LIN {X 79.043,Y 42.209,Z 71.697,A 180.000,B 0.000,C 180.000} C_DIS
LIN {X 79.064,Y 42.285,Z 71.694,A 180.000,B 0.000,C 180.000} C_DIS
LIN {X 79.085,Y 42.362,Z 71.691,A 180.000,B 0.000,C 180.000} C_DIS
LIN {X 79.105,Y 42.438,Z 71.689,A 180.000,B 0.000,C 180.000} C_DIS
LIN {X 79.126,Y 42.514,Z 71.686,A 180.000,B 0.000,C 180.000} C_DIS
LIN {X 79.147,Y 42.590,Z 71.683,A 180.000,B 0.000,C 180.000} C_DIS
LIN {X 79.167,Y 42.666,Z 71.680,A 180.000,B 0.000,C 180.000} C_DIS
LIN {X 79.188,Y 42.742,Z 71.678,A 180.000,B 0.000,C 180.000} C_DIS
LIN {X 79.209,Y 42.818,Z 71.675,A 180.000,B 0.000,C 180.000} C_DIS
LIN {X 79.230,Y 42.894,Z 71.672,A 180.000,B 0.000,C 180.000} C_DIS
LIN {X 79.250,Y 42.971,Z 71.670,A 180.000,B 0.000,C 180.000} C_DIS
LIN {X 79.271,Y 43.047,Z 71.667,A 180.000,B 0.000,C 180.000} C_DIS
LIN {X 79.292,Y 43.123,Z 71.665,A 180.000,B 0.000,C 180.000} C_DIS
LIN {X 79.313,Y 43.199,Z 71.662,A 180.000,B 0.000,C 180.000} C_DIS
LIN {X 79.334,Y 43.275,Z 71.659,A 180.000,B 0.000,C 180.000} C_DIS
LIN {X 79.355,Y 43.351,Z 71.657,A 180.000,B 0.000,C 180.000} C_DIS
LIN {X 79.376,Y 43.427,Z 71.654,A 180.000,B 0.000,C 180.000} C_DIS
LIN {X 79.397,Y 43.503,Z 71.652,A 180.000,B 0.000,C 180.000} C_DIS
LIN {X 79.418,Y 43.579,Z 71.649,A 180.000,B 0.000,C 180.000} C_DIS
LIN {X 79.439,Y 43.655,Z 71.647,A 180.000,B 0.000,C 180.000} C_DIS
LIN {X 79.481,Y 43.807,Z 71.642,A 180.000,B 0.000,C 180.000} C_DIS
LIN {X 79.523,Y 43.959,Z 71.637,A 180.000,B 0.000,C 180.000} C_DIS
LIN {X 79.565,Y 44.111,Z 71.632,A 180.000,B 0.000,C 180.000} C_DIS
LIN {X 79.608,Y 44.263,Z 71.627,A 180.000,B 0.000,C 180.000} C_DIS
LIN {X 79.650,Y 44.415,Z 71.623,A 180.000,B 0.000,C 180.000} C_DIS
LIN {X 79.693,Y 44.566,Z 71.618,A 180.000,B 0.000,C 180.000} C_DIS
LIN {X 79.736,Y 44.718,Z 71.613,A 180.000,B 0.000,C 180.000} C_DIS
LIN {X 79.779,Y 44.870,Z 71.609,A 180.000,B 0.000,C 180.000} C_DIS
LIN {X 79.822,Y 45.022,Z 71.604,A 180.000,B 0.000,C 180.000} C_DIS
LIN {X 79.865,Y 45.173,Z 71.600,A 180.000,B 0.000,C 180.000} C_DIS
LIN {X 79.908,Y 45.325,Z 71.596,A 180.000,B 0.000,C 180.000} C_DIS
LIN {X 79.952,Y 45.477,Z 71.592,A 180.000,B 0.000,C 180.000} C_DIS
LIN {X 79.995,Y 45.628,Z 71.588,A 180.000,B 0.000,C 180.000} C_DIS
LIN {X 80.039,Y 45.780,Z 71.584,A 180.000,B 0.000,C 180.000} C_DIS
LIN {X 80.083,Y 45.931,Z 71.580,A 180.000,B 0.000,C 180.000} C_DIS
LIN {X 80.127,Y 46.082,Z 71.576,A 180.000,B 0.000,C 180.000} C_DIS
LIN {X 80.171,Y 46.234,Z 71.572,A 180.000,B 0.000,C 180.000} C_DIS
LIN {X 80.215,Y 46.385,Z 71.568,A 180.000,B 0.000,C 180.000} C_DIS
LIN {X 80.259,Y 46.536,Z 71.565,A 180.000,B 0.000,C 180.000} C_DIS
LIN {X 80.304,Y 46.688,Z 71.561,A 180.000,B 0.000,C 180.000} C_DIS
LIN {X 80.348,Y 46.839,Z 71.558,A 180.000,B 0.000,C 180.000} C_DIS
LIN {X 80.393,Y 46.990,Z 71.554,A 180.000,B 0.000,C 180.000} C_DIS
LIN {X 80.438,Y 47.141,Z 71.551,A 180.000,B 0.000,C 180.000} C_DIS
LIN {X 80.483,Y 47.292,Z 71.548,A 180.000,B 0.000,C 180.000} C_DIS
LIN {X 80.528,Y 47.443,Z 71.545,A 180.000,B 0.000,C 180.000} C_DIS
LIN {X 80.574,Y 47.594,Z 71.542,A 180.000,B 0.000,C 180.000} C_DIS
LIN {X 80.619,Y 47.745,Z 71.539,A 180.000,B 0.000,C 180.000} C_DIS
LIN {X 80.665,Y 47.895,Z 71.536,A 180.000,B 0.000,C 180.000} C_DIS
LIN {X 80.711,Y 48.046,Z 71.533,A 180.000,B 0.000,C 180.000} C_DIS
LIN {X 80.757,Y 48.197,Z 71.531,A 180.000,B 0.000,C 180.000} C_DIS
LIN {X 80.803,Y 48.348,Z 71.528,A 180.000,B 0.000,C 180.000} C_DIS
LIN {X 80.896,Y 48.649,Z 71.524,A 180.000,B 0.000,C 180.000} C_DIS
LIN {X 80.989,Y 48.950,Z 71.519,A 180.000,B 0.000,C 180.000} C_DIS
LIN {X 81.084,Y 49.250,Z 71.515,A 180.000,B 0.000,C 180.000} C_DIS
LIN {X 81.178,Y 49.551,Z 71.512,A 180.000,B 0.000,C 180.000} C_DIS
LIN {X 81.274,Y 49.851,Z 71.509,A 180.000,B 0.000,C 180.000} C_DIS
LIN {X 81.370,Y 50.151,Z 71.506,A 180.000,B 0.000,C 180.000} C_DIS
LIN {X 81.467,Y 50.451,Z 71.504,A 180.000,B 0.000,C 180.000} C_DIS
LIN {X 81.564,Y 50.750,Z 71.502,A 180.000,B 0.000,C 180.000} C_DIS
LIN {X 81.663,Y 51.049,Z 71.501,A 180.000,B 0.000,C 180.000} C_DIS
LIN {X 81.762,Y 51.348,Z 71.500,A 180.000,B 0.000,C 180.000} C_DIS
LIN {X 81.862,Y 51.647,Z 71.500,A 180.000,B 0.000,C 180.000} C_DIS
LIN {X 81.868,Y 51.663,Z 71.500,A 180.000,B 0.000,C 180.000} C_DIS
; Cutting Move Starts
LIN {X 84.885,Y 60.606,Z 71.500,A 180.000,B 0.000,C 180.000} C_DIS
LIN {X 84.919,Y 60.703,Z 71.500,A 180.000,B 0.000,C 180.000} C_DIS
LIN {X 84.952,Y 60.785,Z 71.500,A 180.000,B 0.000,C 180.000} C_DIS
LIN {X 85.035,Y 60.964,Z 71.500,A 180.000,B 0.000,C 180.000} C_DIS
LIN {X 85.098,Y 61.079,Z 71.500,A 180.000,B 0.000,C 180.000} C_DIS
LIN {X 85.136,Y 61.143,Z 71.500,A 180.000,B 0.000,C 180.000} C_DIS
LIN {X 85.258,Y 61.321,Z 71.500,A 180.000,B 0.000,C 180.000} C_DIS
LIN {X 85.276,Y 61.345,Z 71.500,A 180.000,B 0.000,C 180.000} C_DIS
LIN {X 85.406,Y 61.500,Z 71.500,A 180.000,B 0.000,C 180.000} C_DIS
LIN {X 85.455,Y 61.553,Z 71.500,A 180.000,B 0.000,C 180.000} C_DIS
LIN {X 85.585,Y 61.679,Z 71.500,A 180.000,B 0.000,C 180.000} C_DIS
LIN {X 85.634,Y 61.722,Z 71.500,A 180.000,B 0.000,C 180.000} C_DIS
LIN {X 85.808,Y 61.858,Z 71.500,A 180.000,B 0.000,C 180.000} C_DIS
LIN {X 85.813,Y 61.861,Z 71.500,A 180.000,B 0.000,C 180.000} C_DIS
LIN {X 85.992,Y 61.977,Z 71.500,A 180.000,B 0.000,C 180.000} C_DIS
LIN {X 86.099,Y 62.036,Z 71.500,A 180.000,B 0.000,C 180.000} C_DIS
LIN {X 86.170,Y 62.073,Z 71.500,A 180.000,B 0.000,C 180.000} C_DIS
LIN {X 86.349,Y 62.151,Z 71.500,A 180.000,B 0.000,C 180.000} C_DIS
LIN {X 86.528,Y 62.213,Z 71.500,A 180.000,B 0.000,C 180.000} C_DIS
LIN {X 86.536,Y 62.215,Z 71.500,A 180.000,B 0.000,C 180.000} C_DIS
LIN {X 86.707,Y 62.260,Z 71.500,A 180.000,B 0.000,C 180.000} C_DIS
LIN {X 86.885,Y 62.294,Z 71.500,A 180.000,B 0.000,C 180.000} C_DIS
LIN {X 86.975,Y 62.306,Z 71.500,A 180.000,B 0.000,C 180.000} C_DIS
LIN {X 87.064,Y 62.314,Z 71.500,A 180.000,B 0.000,C 180.000} C_DIS
LIN {X 87.154,Y 62.320,Z 71.500,A 180.000,B 0.000,C 180.000} C_DIS
LIN {X 87.243,Y 62.322,Z 71.500,A 180.000,B 0.000,C 180.000} C_DIS
LIN {X 87.332,Y 62.321,Z 71.500,A 180.000,B 0.000,C 180.000} C_DIS
LIN {X 87.422,Y 62.317,Z 71.500,A 180.000,B 0.000,C 180.000} C_DIS
LIN {X 87.511,Y 62.309,Z 71.500,A 180.000,B 0.000,C 180.000} C_DIS
LIN {X 87.601,Y 62.298,Z 71.500,A 180.000,B 0.000,C 180.000} C_DIS
LIN {X 87.690,Y 62.284,Z 71.500,A 180.000,B 0.000,C 180.000} C_DIS
LIN {X 87.779,Y 62.267,Z 71.500,A 180.000,B 0.000,C 180.000} C_DIS
LIN {X 87.869,Y 62.246,Z 71.500,A 180.000,B 0.000,C 180.000} C_DIS
LIN {X 87.958,Y 62.222,Z 71.500,A 180.000,B 0.000,C 180.000} C_DIS
LIN {X 87.981,Y 62.215,Z 71.500,A 180.000,B 0.000,C 180.000} C_DIS
LIN {X 88.137,Y 62.164,Z 71.500,A 180.000,B 0.000,C 180.000} C_DIS
LIN {X 96.464,Y 59.355,Z 71.500,A 180.000,B 0.000,C 180.000} C_DIS
LIN {X 96.539,Y 59.329,Z 71.500,A 180.000,B 0.000,C 180.000} C_DIS
LIN {X 96.718,Y 59.257,Z 71.500,A 180.000,B 0.000,C 180.000} C_DIS
LIN {X 96.883,Y 59.176,Z 71.500,A 180.000,B 0.000,C 180.000} C_DIS
LIN {X 96.897,Y 59.169,Z 71.500,A 180.000,B 0.000,C 180.000} C_DIS
LIN {X 97.075,Y 59.061,Z 71.500,A 180.000,B 0.000,C 180.000} C_DIS
LIN {X 97.167,Y 58.997,Z 71.500,A 180.000,B 0.000,C 180.000} C_DIS
LIN {X 97.254,Y 58.931,Z 71.500,A 180.000,B 0.000,C 180.000} C_DIS
LIN {X 97.385,Y 58.819,Z 71.500,A 180.000,B 0.000,C 180.000} C_DIS
LIN {X 97.433,Y 58.774,Z 71.500,A 180.000,B 0.000,C 180.000} C_DIS
LIN {X 97.562,Y 58.640,Z 71.500,A 180.000,B 0.000,C 180.000} C_DIS
LIN {X 97.612,Y 58.582,Z 71.500,A 180.000,B 0.000,C 180.000} C_DIS
LIN {X 97.707,Y 58.461,Z 71.500,A 180.000,B 0.000,C 180.000} C_DIS
LIN {X 97.790,Y 58.341,Z 71.500,A 180.000,B 0.000,C 180.000} C_DIS
LIN {X 97.828,Y 58.282,Z 71.500,A 180.000,B 0.000,C 180.000} C_DIS
LIN {X 97.928,Y 58.103,Z 71.500,A 180.000,B 0.000,C 180.000} C_DIS
LIN {X 97.969,Y 58.017,Z 71.500,A 180.000,B 0.000,C 180.000} C_DIS
LIN {X 98.009,Y 57.925,Z 71.500,A 180.000,B 0.000,C 180.000} C_DIS
LIN {X 98.075,Y 57.746,Z 71.500,A 180.000,B 0.000,C 180.000} C_DIS
LIN {X 98.125,Y 57.567,Z 71.500,A 180.000,B 0.000,C 180.000} C_DIS
LIN {X 98.148,Y 57.466,Z 71.500,A 180.000,B 0.000,C 180.000} C_DIS
LIN {X 98.162,Y 57.388,Z 71.500,A 180.000,B 0.000,C 180.000} C_DIS
LIN {X 98.186,Y 57.210,Z 71.500,A 180.000,B 0.000,C 180.000} C_DIS
LIN {X 98.196,Y 57.031,Z 71.500,A 180.000,B 0.000,C 180.000} C_DIS
LIN {X 98.193,Y 56.852,Z 71.500,A 180.000,B 0.000,C 180.000} C_DIS
LIN {X 98.178,Y 56.673,Z 71.500,A 180.000,B 0.000,C 180.000} C_DIS
LIN {X 98.150,Y 56.495,Z 71.500,A 180.000,B 0.000,C 180.000} C_DIS
LIN {X 98.148,Y 56.485,Z 71.500,A 180.000,B 0.000,C 180.000} C_DIS
LIN {X 98.108,Y 56.316,Z 71.500,A 180.000,B 0.000,C 180.000} C_DIS
LIN {X 98.052,Y 56.137,Z 71.500,A 180.000,B 0.000,C 180.000} C_DIS
LIN {X 91.712,Y 37.344,Z 71.500,A 180.000,B 0.000,C 180.000} C_DIS
LIN {X 91.659,Y 37.187,Z 71.500,A 180.000,B 0.000,C 180.000} C_DIS
LIN {X 91.588,Y 37.009,Z 71.500,A 180.000,B 0.000,C 180.000} C_DIS
LIN {X 91.533,Y 36.894,Z 71.500,A 180.000,B 0.000,C 180.000} C_DIS
LIN {X 91.500,Y 36.830,Z 71.500,A 180.000,B 0.000,C 180.000} C_DIS
LIN {X 91.392,Y 36.651,Z 71.500,A 180.000,B 0.000,C 180.000} C_DIS
LIN {X 91.355,Y 36.595,Z 71.500,A 180.000,B 0.000,C 180.000} C_DIS
LIN {X 91.263,Y 36.472,Z 71.500,A 180.000,B 0.000,C 180.000} C_DIS
LIN {X 91.176,Y 36.368,Z 71.500,A 180.000,B 0.000,C 180.000} C_DIS
LIN {X 91.107,Y 36.294,Z 71.500,A 180.000,B 0.000,C 180.000} C_DIS
LIN {X 90.997,Y 36.186,Z 71.500,A 180.000,B 0.000,C 180.000} C_DIS
LIN {X 90.917,Y 36.115,Z 71.500,A 180.000,B 0.000,C 180.000} C_DIS
LIN {X 90.818,Y 36.036,Z 71.500,A 180.000,B 0.000,C 180.000} C_DIS
LIN {X 90.677,Y 35.936,Z 71.500,A 180.000,B 0.000,C 180.000} C_DIS
LIN {X 90.640,Y 35.912,Z 71.500,A 180.000,B 0.000,C 180.000} C_DIS
LIN {X 90.461,Y 35.809,Z 71.500,A 180.000,B 0.000,C 180.000} C_DIS
LIN {X 90.356,Y 35.757,Z 71.500,A 180.000,B 0.000,C 180.000} C_DIS
LIN {X 90.282,Y 35.724,Z 71.500,A 180.000,B 0.000,C 180.000} C_DIS
LIN {X 90.103,Y 35.656,Z 71.500,A 180.000,B 0.000,C 180.000} C_DIS
LIN {X 89.925,Y 35.603,Z 71.500,A 180.000,B 0.000,C 180.000} C_DIS
LIN {X 89.819,Y 35.578,Z 71.500,A 180.000,B 0.000,C 180.000} C_DIS
LIN {X 89.746,Y 35.564,Z 71.500,A 180.000,B 0.000,C 180.000} C_DIS
LIN {X 89.567,Y 35.539,Z 71.500,A 180.000,B 0.000,C 180.000} C_DIS
LIN {X 89.388,Y 35.526,Z 71.500,A 180.000,B 0.000,C 180.000} C_DIS
LIN {X 89.209,Y 35.526,Z 71.500,A 180.000,B 0.000,C 180.000} C_DIS
LIN {X 89.031,Y 35.540,Z 71.500,A 180.000,B 0.000,C 180.000} C_DIS
LIN {X 88.852,Y 35.566,Z 71.500,A 180.000,B 0.000,C 180.000} C_DIS
LIN {X 88.788,Y 35.578,Z 71.500,A 180.000,B 0.000,C 180.000} C_DIS
LIN {X 88.673,Y 35.605,Z 71.500,A 180.000,B 0.000,C 180.000} C_DIS
LIN {X 88.494,Y 35.659,Z 71.500,A 180.000,B 0.000,C 180.000} C_DIS
LIN {X 80.092,Y 38.494,Z 71.500,A 180.000,B 0.000,C 180.000} C_DIS
LIN {X 80.003,Y 38.525,Z 71.500,A 180.000,B 0.000,C 180.000} C_DIS
LIN {X 79.913,Y 38.560,Z 71.500,A 180.000,B 0.000,C 180.000} C_DIS
LIN {X 79.848,Y 38.587,Z 71.500,A 180.000,B 0.000,C 180.000} C_DIS
LIN {X 79.783,Y 38.618,Z 71.500,A 180.000,B 0.000,C 180.000} C_DIS
LIN {X 79.735,Y 38.642,Z 71.500,A 180.000,B 0.000,C 180.000} C_DIS
LIN {X 79.645,Y 38.689,Z 71.500,A 180.000,B 0.000,C 180.000} C_DIS
LIN {X 79.556,Y 38.742,Z 71.500,A 180.000,B 0.000,C 180.000} C_DIS
LIN {X 79.471,Y 38.796,Z 71.500,A 180.000,B 0.000,C 180.000} C_DIS
LIN {X 79.377,Y 38.863,Z 71.500,A 180.000,B 0.000,C 180.000} C_DIS
LIN {X 79.307,Y 38.917,Z 71.500,A 180.000,B 0.000,C 180.000} C_DIS
LIN {X 79.236,Y 38.975,Z 71.500,A 180.000,B 0.000,C 180.000} C_DIS
LIN {X 79.198,Y 39.008,Z 71.500,A 180.000,B 0.000,C 180.000} C_DIS
LIN {X 79.124,Y 39.078,Z 71.500,A 180.000,B 0.000,C 180.000} C_DIS
LIN {X 79.049,Y 39.154,Z 71.500,A 180.000,B 0.000,C 180.000} C_DIS
LIN {X 79.020,Y 39.185,Z 71.500,A 180.000,B 0.000,C 180.000} C_DIS
LIN {X 78.895,Y 39.333,Z 71.500,A 180.000,B 0.000,C 180.000} C_DIS
LIN {X 78.841,Y 39.405,Z 71.500,A 180.000,B 0.000,C 180.000} C_DIS
LIN {X 78.768,Y 39.511,Z 71.500,A 180.000,B 0.000,C 180.000} C_DIS
LIN {X 78.662,Y 39.690,Z 71.500,A 180.000,B 0.000,C 180.000} C_DIS
LIN {X 78.662,Y 39.690,Z 71.500,A 180.000,B 0.000,C 180.000} C_DIS
LIN {X 78.575,Y 39.869,Z 71.500,A 180.000,B 0.000,C 180.000} C_DIS
LIN {X 78.505,Y 40.048,Z 71.500,A 180.000,B 0.000,C 180.000} C_DIS
LIN {X 78.483,Y 40.113,Z 71.500,A 180.000,B 0.000,C 180.000} C_DIS
LIN {X 78.450,Y 40.226,Z 71.500,A 180.000,B 0.000,C 180.000} C_DIS
LIN {X 78.409,Y 40.405,Z 71.500,A 180.000,B 0.000,C 180.000} C_DIS
LIN {X 78.382,Y 40.584,Z 71.500,A 180.000,B 0.000,C 180.000} C_DIS
LIN {X 78.368,Y 40.763,Z 71.500,A 180.000,B 0.000,C 180.000} C_DIS
LIN {X 78.367,Y 40.942,Z 71.500,A 180.000,B 0.000,C 180.000} C_DIS
LIN {X 78.378,Y 41.120,Z 71.500,A 180.000,B 0.000,C 180.000} C_DIS
LIN {X 78.403,Y 41.299,Z 71.500,A 180.000,B 0.000,C 180.000} C_DIS
LIN {X 78.440,Y 41.478,Z 71.500,A 180.000,B 0.000,C 180.000} C_DIS
LIN {X 78.483,Y 41.629,Z 71.500,A 180.000,B 0.000,C 180.000} C_DIS
LIN {X 78.492,Y 41.657,Z 71.500,A 180.000,B 0.000,C 180.000} C_DIS
LIN {X 78.552,Y 41.835,Z 71.500,A 180.000,B 0.000,C 180.000} C_DIS
LIN {X 81.868,Y 51.663,Z 71.500,A 180.000,B 0.000,C 180.000} C_DIS
; Link Move Starts
LIN {X 81.968,Y 51.961,Z 71.500,A 180.000,B 0.000,C 180.000} C_DIS
LIN {X 82.067,Y 52.260,Z 71.499,A 180.000,B 0.000,C 180.000} C_DIS
LIN {X 82.166,Y 52.560,Z 71.498,A 180.000,B 0.000,C 180.000} C_DIS
LIN {X 82.264,Y 52.859,Z 71.496,A 180.000,B 0.000,C 180.000} C_DIS
LIN {X 82.361,Y 53.159,Z 71.494,A 180.000,B 0.000,C 180.000} C_DIS
LIN {X 82.457,Y 53.459,Z 71.491,A 180.000,B 0.000,C 180.000} C_DIS
LIN {X 82.552,Y 53.759,Z 71.488,A 180.000,B 0.000,C 180.000} C_DIS
LIN {X 82.647,Y 54.060,Z 71.485,A 180.000,B 0.000,C 180.000} C_DIS
LIN {X 82.740,Y 54.360,Z 71.481,A 180.000,B 0.000,C 180.000} C_DIS
LIN {X 82.833,Y 54.662,Z 71.477,A 180.000,B 0.000,C 180.000} C_DIS
LIN {X 82.926,Y 54.963,Z 71.472,A 180.000,B 0.000,C 180.000} C_DIS
LIN {X 82.972,Y 55.114,Z 71.469,A 180.000,B 0.000,C 180.000} C_DIS
LIN {X 83.017,Y 55.264,Z 71.467,A 180.000,B 0.000,C 180.000} C_DIS
LIN {X 83.063,Y 55.415,Z 71.464,A 180.000,B 0.000,C 180.000} C_DIS
LIN {X 83.108,Y 55.566,Z 71.461,A 180.000,B 0.000,C 180.000} C_DIS
LIN {X 83.154,Y 55.717,Z 71.459,A 180.000,B 0.000,C 180.000} C_DIS
LIN {X 83.199,Y 55.868,Z 71.456,A 180.000,B 0.000,C 180.000} C_DIS
LIN {X 83.243,Y 56.019,Z 71.452,A 180.000,B 0.000,C 180.000} C_DIS
LIN {X 83.288,Y 56.170,Z 71.449,A 180.000,B 0.000,C 180.000} C_DIS
LIN {X 83.333,Y 56.321,Z 71.446,A 180.000,B 0.000,C 180.000} C_DIS
LIN {X 83.377,Y 56.473,Z 71.443,A 180.000,B 0.000,C 180.000} C_DIS
LIN {X 83.421,Y 56.624,Z 71.439,A 180.000,B 0.000,C 180.000} C_DIS
LIN {X 83.466,Y 56.775,Z 71.436,A 180.000,B 0.000,C 180.000} C_DIS
LIN {X 83.510,Y 56.927,Z 71.432,A 180.000,B 0.000,C 180.000} C_DIS
LIN {X 83.553,Y 57.078,Z 71.428,A 180.000,B 0.000,C 180.000} C_DIS
LIN {X 83.597,Y 57.230,Z 71.425,A 180.000,B 0.000,C 180.000} C_DIS
LIN {X 83.640,Y 57.381,Z 71.421,A 180.000,B 0.000,C 180.000} C_DIS
LIN {X 83.684,Y 57.533,Z 71.417,A 180.000,B 0.000,C 180.000} C_DIS
LIN {X 83.727,Y 57.684,Z 71.413,A 180.000,B 0.000,C 180.000} C_DIS
LIN {X 83.770,Y 57.836,Z 71.409,A 180.000,B 0.000,C 180.000} C_DIS
LIN {X 83.813,Y 57.988,Z 71.405,A 180.000,B 0.000,C 180.000} C_DIS
LIN {X 83.856,Y 58.140,Z 71.400,A 180.000,B 0.000,C 180.000} C_DIS
LIN {X 83.899,Y 58.291,Z 71.396,A 180.000,B 0.000,C 180.000} C_DIS
LIN {X 83.941,Y 58.443,Z 71.392,A 180.000,B 0.000,C 180.000} C_DIS
LIN {X 83.984,Y 58.595,Z 71.387,A 180.000,B 0.000,C 180.000} C_DIS
LIN {X 84.026,Y 58.747,Z 71.383,A 180.000,B 0.000,C 180.000} C_DIS
LIN {X 84.068,Y 58.899,Z 71.378,A 180.000,B 0.000,C 180.000} C_DIS
LIN {X 84.110,Y 59.051,Z 71.373,A 180.000,B 0.000,C 180.000} C_DIS
LIN {X 84.152,Y 59.203,Z 71.369,A 180.000,B 0.000,C 180.000} C_DIS
LIN {X 84.194,Y 59.355,Z 71.364,A 180.000,B 0.000,C 180.000} C_DIS
LIN {X 84.235,Y 59.508,Z 71.359,A 180.000,B 0.000,C 180.000} C_DIS
LIN {X 84.277,Y 59.660,Z 71.354,A 180.000,B 0.000,C 180.000} C_DIS
LIN {X 84.298,Y 59.736,Z 71.351,A 180.000,B 0.000,C 180.000} C_DIS
LIN {X 84.318,Y 59.812,Z 71.349,A 180.000,B 0.000,C 180.000} C_DIS
LIN {X 84.339,Y 59.888,Z 71.346,A 180.000,B 0.000,C 180.000} C_DIS
LIN {X 84.360,Y 59.964,Z 71.344,A 180.000,B 0.000,C 180.000} C_DIS
LIN {X 84.380,Y 60.040,Z 71.341,A 180.000,B 0.000,C 180.000} C_DIS
LIN {X 84.401,Y 60.117,Z 71.339,A 180.000,B 0.000,C 180.000} C_DIS
LIN {X 84.422,Y 60.193,Z 71.336,A 180.000,B 0.000,C 180.000} C_DIS
LIN {X 84.442,Y 60.269,Z 71.333,A 180.000,B 0.000,C 180.000} C_DIS
LIN {X 84.463,Y 60.345,Z 71.331,A 180.000,B 0.000,C 180.000} C_DIS
LIN {X 84.483,Y 60.421,Z 71.328,A 180.000,B 0.000,C 180.000} C_DIS
LIN {X 84.518,Y 60.553,Z 71.323,A 180.000,B 0.000,C 180.000} C_DIS
LIN {X 84.553,Y 60.684,Z 71.319,A 180.000,B 0.000,C 180.000} C_DIS
LIN {X 84.581,Y 60.787,Z 71.315,A 180.000,B 0.000,C 180.000} C_DIS
LIN {X 84.604,Y 60.864,Z 71.312,A 180.000,B 0.000,C 180.000} C_DIS
LIN {X 84.624,Y 60.924,Z 71.310,A 180.000,B 0.000,C 180.000} C_DIS
LIN {X 84.653,Y 61.001,Z 71.307,A 180.000,B 0.000,C 180.000} C_DIS
LIN {X 84.685,Y 61.079,Z 71.304,A 180.000,B 0.000,C 180.000} C_DIS
LIN {X 84.727,Y 61.173,Z 71.301,A 180.000,B 0.000,C 180.000} C_DIS
LIN {X 84.789,Y 61.294,Z 71.296,A 180.000,B 0.000,C 180.000} C_DIS
LIN {X 84.847,Y 61.392,Z 71.292,A 180.000,B 0.000,C 180.000} C_DIS
LIN {X 84.898,Y 61.471,Z 71.289,A 180.000,B 0.000,C 180.000} C_DIS
LIN {X 84.952,Y 61.548,Z 71.286,A 180.000,B 0.000,C 180.000} C_DIS
LIN {X 85.010,Y 61.623,Z 71.283,A 180.000,B 0.000,C 180.000} C_DIS
LIN {X 85.070,Y 61.696,Z 71.280,A 180.000,B 0.000,C 180.000} C_DIS
LIN {X 85.152,Y 61.785,Z 71.277,A 180.000,B 0.000,C 180.000} C_DIS
LIN {X 85.238,Y 61.870,Z 71.273,A 180.000,B 0.000,C 180.000} C_DIS
LIN {X 85.347,Y 61.967,Z 71.268,A 180.000,B 0.000,C 180.000} C_DIS
LIN {X 85.462,Y 62.056,Z 71.264,A 180.000,B 0.000,C 180.000} C_DIS
LIN {X 85.543,Y 62.114,Z 71.260,A 180.000,B 0.000,C 180.000} C_DIS
LIN {X 85.627,Y 62.167,Z 71.257,A 180.000,B 0.000,C 180.000} C_DIS
LIN {X 85.713,Y 62.217,Z 71.253,A 180.000,B 0.000,C 180.000} C_DIS
LIN {X 85.801,Y 62.263,Z 71.250,A 180.000,B 0.000,C 180.000} C_DIS
LIN {X 85.894,Y 62.307,Z 71.246,A 180.000,B 0.000,C 180.000} C_DIS
LIN {X 85.989,Y 62.346,Z 71.243,A 180.000,B 0.000,C 180.000} C_DIS
LIN {X 86.085,Y 62.381,Z 71.239,A 180.000,B 0.000,C 180.000} C_DIS
LIN {X 86.183,Y 62.412,Z 71.235,A 180.000,B 0.000,C 180.000} C_DIS
LIN {X 86.271,Y 62.435,Z 71.232,A 180.000,B 0.000,C 180.000} C_DIS
LIN {X 86.360,Y 62.454,Z 71.229,A 180.000,B 0.000,C 180.000} C_DIS
LIN {X 86.449,Y 62.470,Z 71.226,A 180.000,B 0.000,C 180.000} C_DIS
LIN {X 86.540,Y 62.483,Z 71.223,A 180.000,B 0.000,C 180.000} C_DIS
LIN {X 86.623,Y 62.491,Z 71.220,A 180.000,B 0.000,C 180.000} C_DIS
LIN {X 86.708,Y 62.495,Z 71.217,A 180.000,B 0.000,C 180.000} C_DIS
LIN {X 86.792,Y 62.497,Z 71.214,A 180.000,B 0.000,C 180.000} C_DIS
LIN {X 86.876,Y 62.495,Z 71.211,A 180.000,B 0.000,C 180.000} C_DIS
LIN {X 86.957,Y 62.491,Z 71.208,A 180.000,B 0.000,C 180.000} C_DIS
LIN {X 87.037,Y 62.483,Z 71.205,A 180.000,B 0.000,C 180.000} C_DIS
LIN {X 87.117,Y 62.473,Z 71.203,A 180.000,B 0.000,C 180.000} C_DIS
LIN {X 87.196,Y 62.459,Z 71.200,A 180.000,B 0.000,C 180.000} C_DIS
LIN {X 87.274,Y 62.443,Z 71.197,A 180.000,B 0.000,C 180.000} C_DIS
LIN {X 87.351,Y 62.424,Z 71.194,A 180.000,B 0.000,C 180.000} C_DIS
LIN {X 87.427,Y 62.403,Z 71.191,A 180.000,B 0.000,C 180.000} C_DIS
LIN {X 87.502,Y 62.378,Z 71.189,A 180.000,B 0.000,C 180.000} C_DIS
LIN {X 87.651,Y 62.328,Z 71.183,A 180.000,B 0.000,C 180.000} C_DIS
LIN {X 88.099,Y 62.177,Z 71.167,A 180.000,B 0.000,C 180.000} C_DIS
LIN {X 88.322,Y 62.101,Z 71.158,A 180.000,B 0.000,C 180.000} C_DIS
LIN {X 88.472,Y 62.051,Z 71.153,A 180.000,B 0.000,C 180.000} C_DIS
LIN {X 88.919,Y 61.900,Z 71.136,A 180.000,B 0.000,C 180.000} C_DIS
LIN {X 89.069,Y 61.850,Z 71.131,A 180.000,B 0.000,C 180.000} C_DIS
LIN {X 89.516,Y 61.699,Z 71.114,A 180.000,B 0.000,C 180.000} C_DIS
LIN {X 89.666,Y 61.648,Z 71.109,A 180.000,B 0.000,C 180.000} C_DIS
LIN {X 90.337,Y 61.422,Z 71.084,A 180.000,B 0.000,C 180.000} C_DIS
LIN {X 91.382,Y 61.069,Z 71.046,A 180.000,B 0.000,C 180.000} C_DIS
LIN {X 92.053,Y 60.843,Z 71.021,A 180.000,B 0.000,C 180.000} C_DIS
LIN {X 96.456,Y 59.358,Z 70.859,A 180.000,B 0.000,C 180.000} C_DIS
LIN {X 96.530,Y 59.332,Z 70.856,A 180.000,B 0.000,C 180.000} C_DIS
LIN {X 96.604,Y 59.305,Z 70.853,A 180.000,B 0.000,C 180.000} C_DIS
LIN {X 96.677,Y 59.275,Z 70.850,A 180.000,B 0.000,C 180.000} C_DIS
LIN {X 96.749,Y 59.243,Z 70.848,A 180.000,B 0.000,C 180.000} C_DIS
LIN {X 96.820,Y 59.209,Z 70.845,A 180.000,B 0.000,C 180.000} C_DIS
LIN {X 96.890,Y 59.172,Z 70.842,A 180.000,B 0.000,C 180.000} C_DIS
LIN {X 96.958,Y 59.133,Z 70.839,A 180.000,B 0.000,C 180.000} C_DIS
LIN {X 97.026,Y 59.093,Z 70.837,A 180.000,B 0.000,C 180.000} C_DIS
LIN {X 97.092,Y 59.050,Z 70.834,A 180.000,B 0.000,C 180.000} C_DIS
LIN {X 97.156,Y 59.005,Z 70.831,A 180.000,B 0.000,C 180.000} C_DIS
LIN {X 97.220,Y 58.958,Z 70.828,A 180.000,B 0.000,C 180.000} C_DIS
LIN {X 97.281,Y 58.909,Z 70.826,A 180.000,B 0.000,C 180.000} C_DIS
LIN {X 97.341,Y 58.858,Z 70.823,A 180.000,B 0.000,C 180.000} C_DIS
LIN {X 97.400,Y 58.805,Z 70.820,A 180.000,B 0.000,C 180.000} C_DIS
LIN {X 97.457,Y 58.751,Z 70.817,A 180.000,B 0.000,C 180.000} C_DIS
LIN {X 97.512,Y 58.694,Z 70.815,A 180.000,B 0.000,C 180.000} C_DIS
LIN {X 97.565,Y 58.636,Z 70.812,A 180.000,B 0.000,C 180.000} C_DIS
LIN {X 97.616,Y 58.577,Z 70.809,A 180.000,B 0.000,C 180.000} C_DIS
LIN {X 97.666,Y 58.515,Z 70.806,A 180.000,B 0.000,C 180.000} C_DIS
LIN {X 97.713,Y 58.452,Z 70.804,A 180.000,B 0.000,C 180.000} C_DIS
LIN {X 97.759,Y 58.388,Z 70.801,A 180.000,B 0.000,C 180.000} C_DIS
LIN {X 97.802,Y 58.323,Z 70.798,A 180.000,B 0.000,C 180.000} C_DIS
LIN {X 97.844,Y 58.256,Z 70.795,A 180.000,B 0.000,C 180.000} C_DIS
LIN {X 97.883,Y 58.187,Z 70.793,A 180.000,B 0.000,C 180.000} C_DIS
LIN {X 97.920,Y 58.118,Z 70.790,A 180.000,B 0.000,C 180.000} C_DIS
LIN {X 97.955,Y 58.047,Z 70.787,A 180.000,B 0.000,C 180.000} C_DIS
LIN {X 97.988,Y 57.976,Z 70.784,A 180.000,B 0.000,C 180.000} C_DIS
LIN {X 98.018,Y 57.903,Z 70.782,A 180.000,B 0.000,C 180.000} C_DIS
LIN {X 98.046,Y 57.829,Z 70.779,A 180.000,B 0.000,C 180.000} C_DIS
LIN {X 98.072,Y 57.755,Z 70.776,A 180.000,B 0.000,C 180.000} C_DIS
LIN {X 98.095,Y 57.680,Z 70.773,A 180.000,B 0.000,C 180.000} C_DIS
LIN {X 98.116,Y 57.604,Z 70.771,A 180.000,B 0.000,C 180.000} C_DIS
LIN {X 98.135,Y 57.527,Z 70.768,A 180.000,B 0.000,C 180.000} C_DIS
LIN {X 98.151,Y 57.450,Z 70.765,A 180.000,B 0.000,C 180.000} C_DIS
LIN {X 98.165,Y 57.373,Z 70.763,A 180.000,B 0.000,C 180.000} C_DIS
LIN {X 98.176,Y 57.295,Z 70.760,A 180.000,B 0.000,C 180.000} C_DIS
LIN {X 98.185,Y 57.216,Z 70.757,A 180.000,B 0.000,C 180.000} C_DIS
LIN {X 98.191,Y 57.138,Z 70.754,A 180.000,B 0.000,C 180.000} C_DIS
LIN {X 98.195,Y 57.059,Z 70.752,A 180.000,B 0.000,C 180.000} C_DIS
LIN {X 98.196,Y 56.980,Z 70.749,A 180.000,B 0.000,C 180.000} C_DIS
LIN {X 98.195,Y 56.902,Z 70.746,A 180.000,B 0.000,C 180.000} C_DIS
LIN {X 98.192,Y 56.823,Z 70.743,A 180.000,B 0.000,C 180.000} C_DIS
LIN {X 98.186,Y 56.744,Z 70.741,A 180.000,B 0.000,C 180.000} C_DIS
LIN {X 98.177,Y 56.666,Z 70.738,A 180.000,B 0.000,C 180.000} C_DIS
LIN {X 98.166,Y 56.588,Z 70.735,A 180.000,B 0.000,C 180.000} C_DIS
LIN {X 98.153,Y 56.511,Z 70.732,A 180.000,B 0.000,C 180.000} C_DIS
LIN {X 98.137,Y 56.433,Z 70.730,A 180.000,B 0.000,C 180.000} C_DIS
LIN {X 98.119,Y 56.357,Z 70.727,A 180.000,B 0.000,C 180.000} C_DIS
LIN {X 98.098,Y 56.281,Z 70.724,A 180.000,B 0.000,C 180.000} C_DIS
LIN {X 98.075,Y 56.205,Z 70.721,A 180.000,B 0.000,C 180.000} C_DIS
LIN {X 98.050,Y 56.131,Z 70.719,A 180.000,B 0.000,C 180.000} C_DIS
LIN {X 98.025,Y 56.056,Z 70.716,A 180.000,B 0.000,C 180.000} C_DIS
LIN {X 97.974,Y 55.907,Z 70.710,A 180.000,B 0.000,C 180.000} C_DIS
LIN {X 97.899,Y 55.683,Z 70.702,A 180.000,B 0.000,C 180.000} C_DIS
LIN {X 97.849,Y 55.534,Z 70.697,A 180.000,B 0.000,C 180.000} C_DIS
LIN {X 97.823,Y 55.459,Z 70.694,A 180.000,B 0.000,C 180.000} C_DIS
LIN {X 97.773,Y 55.310,Z 70.688,A 180.000,B 0.000,C 180.000} C_DIS
LIN {X 97.723,Y 55.161,Z 70.683,A 180.000,B 0.000,C 180.000} C_DIS
LIN {X 97.672,Y 55.011,Z 70.677,A 180.000,B 0.000,C 180.000} C_DIS
LIN {X 97.622,Y 54.862,Z 70.672,A 180.000,B 0.000,C 180.000} C_DIS
LIN {X 97.572,Y 54.713,Z 70.667,A 180.000,B 0.000,C 180.000} C_DIS
LIN {X 97.547,Y 54.638,Z 70.664,A 180.000,B 0.000,C 180.000} C_DIS
LIN {X 97.521,Y 54.564,Z 70.662,A 180.000,B 0.000,C 180.000} C_DIS
LIN {X 97.496,Y 54.489,Z 70.659,A 180.000,B 0.000,C 180.000} C_DIS
LIN {X 97.471,Y 54.415,Z 70.657,A 180.000,B 0.000,C 180.000} C_DIS
LIN {X 97.446,Y 54.340,Z 70.654,A 180.000,B 0.000,C 180.000} C_DIS
LIN {X 97.421,Y 54.265,Z 70.651,A 180.000,B 0.000,C 180.000} C_DIS
LIN {X 97.396,Y 54.191,Z 70.649,A 180.000,B 0.000,C 180.000} C_DIS
LIN {X 97.370,Y 54.116,Z 70.646,A 180.000,B 0.000,C 180.000} C_DIS
LIN {X 97.320,Y 53.967,Z 70.641,A 180.000,B 0.000,C 180.000} C_DIS
LIN {X 97.270,Y 53.818,Z 70.637,A 180.000,B 0.000,C 180.000} C_DIS
LIN {X 97.219,Y 53.668,Z 70.632,A 180.000,B 0.000,C 180.000} C_DIS
LIN {X 97.169,Y 53.519,Z 70.627,A 180.000,B 0.000,C 180.000} C_DIS
LIN {X 97.119,Y 53.370,Z 70.622,A 180.000,B 0.000,C 180.000} C_DIS
LIN {X 97.068,Y 53.221,Z 70.618,A 180.000,B 0.000,C 180.000} C_DIS
LIN {X 97.018,Y 53.071,Z 70.613,A 180.000,B 0.000,C 180.000} C_DIS
LIN {X 96.968,Y 52.922,Z 70.609,A 180.000,B 0.000,C 180.000} C_DIS
LIN {X 96.917,Y 52.773,Z 70.604,A 180.000,B 0.000,C 180.000} C_DIS
LIN {X 96.867,Y 52.624,Z 70.600,A 180.000,B 0.000,C 180.000} C_DIS
LIN {X 96.817,Y 52.474,Z 70.596,A 180.000,B 0.000,C 180.000} C_DIS
LIN {X 96.766,Y 52.325,Z 70.591,A 180.000,B 0.000,C 180.000} C_DIS
LIN {X 96.716,Y 52.176,Z 70.587,A 180.000,B 0.000,C 180.000} C_DIS
LIN {X 96.666,Y 52.027,Z 70.583,A 180.000,B 0.000,C 180.000} C_DIS
LIN {X 96.615,Y 51.878,Z 70.579,A 180.000,B 0.000,C 180.000} C_DIS
LIN {X 96.565,Y 51.728,Z 70.576,A 180.000,B 0.000,C 180.000} C_DIS
LIN {X 96.514,Y 51.579,Z 70.572,A 180.000,B 0.000,C 180.000} C_DIS
LIN {X 96.464,Y 51.430,Z 70.568,A 180.000,B 0.000,C 180.000} C_DIS
LIN {X 96.414,Y 51.281,Z 70.564,A 180.000,B 0.000,C 180.000} C_DIS
LIN {X 96.363,Y 51.131,Z 70.561,A 180.000,B 0.000,C 180.000} C_DIS
LIN {X 96.313,Y 50.982,Z 70.557,A 180.000,B 0.000,C 180.000} C_DIS
LIN {X 96.263,Y 50.833,Z 70.554,A 180.000,B 0.000,C 180.000} C_DIS
LIN {X 96.212,Y 50.684,Z 70.551,A 180.000,B 0.000,C 180.000} C_DIS
LIN {X 96.162,Y 50.534,Z 70.548,A 180.000,B 0.000,C 180.000} C_DIS
LIN {X 96.112,Y 50.385,Z 70.545,A 180.000,B 0.000,C 180.000} C_DIS
LIN {X 96.061,Y 50.236,Z 70.542,A 180.000,B 0.000,C 180.000} C_DIS
LIN {X 96.011,Y 50.087,Z 70.539,A 180.000,B 0.000,C 180.000} C_DIS
LIN {X 95.961,Y 49.937,Z 70.536,A 180.000,B 0.000,C 180.000} C_DIS
LIN {X 95.910,Y 49.788,Z 70.533,A 180.000,B 0.000,C 180.000} C_DIS
LIN {X 95.860,Y 49.639,Z 70.531,A 180.000,B 0.000,C 180.000} C_DIS
LIN {X 95.810,Y 49.490,Z 70.528,A 180.000,B 0.000,C 180.000} C_DIS
LIN {X 95.709,Y 49.191,Z 70.523,A 180.000,B 0.000,C 180.000} C_DIS
LIN {X 95.608,Y 48.893,Z 70.519,A 180.000,B 0.000,C 180.000} C_DIS
LIN {X 95.508,Y 48.594,Z 70.515,A 180.000,B 0.000,C 180.000} C_DIS
LIN {X 95.407,Y 48.296,Z 70.512,A 180.000,B 0.000,C 180.000} C_DIS
LIN {X 95.306,Y 47.997,Z 70.509,A 180.000,B 0.000,C 180.000} C_DIS
LIN {X 95.206,Y 47.699,Z 70.506,A 180.000,B 0.000,C 180.000} C_DIS
LIN {X 95.105,Y 47.400,Z 70.504,A 180.000,B 0.000,C 180.000} C_DIS
LIN {X 95.004,Y 47.102,Z 70.502,A 180.000,B 0.000,C 180.000} C_DIS
LIN {X 94.903,Y 46.803,Z 70.501,A 180.000,B 0.000,C 180.000} C_DIS
LIN {X 94.803,Y 46.505,Z 70.500,A 180.000,B 0.000,C 180.000} C_DIS
LIN {X 94.699,Y 46.199,Z 70.500,A 180.000,B 0.000,C 180.000} C_DIS
; Cutting Move Starts
LIN {X 91.712,Y 37.344,Z 70.500,A 180.000,B 0.000,C 180.000} C_DIS
LIN {X 91.659,Y 37.187,Z 70.500,A 180.000,B 0.000,C 180.000} C_DIS
LIN {X 91.588,Y 37.009,Z 70.500,A 180.000,B 0.000,C 180.000} C_DIS
LIN {X 91.533,Y 36.894,Z 70.500,A 180.000,B 0.000,C 180.000} C_DIS
LIN {X 91.500,Y 36.830,Z 70.500,A 180.000,B 0.000,C 180.000} C_DIS
LIN {X 91.392,Y 36.651,Z 70.500,A 180.000,B 0.000,C 180.000} C_DIS
LIN {X 91.355,Y 36.595,Z 70.500,A 180.000,B 0.000,C 180.000} C_DIS
LIN {X 91.263,Y 36.472,Z 70.500,A 180.000,B 0.000,C 180.000} C_DIS
LIN {X 91.176,Y 36.368,Z 70.500,A 180.000,B 0.000,C 180.000} C_DIS
LIN {X 91.107,Y 36.294,Z 70.500,A 180.000,B 0.000,C 180.000} C_DIS
LIN {X 90.997,Y 36.186,Z 70.500,A 180.000,B 0.000,C 180.000} C_DIS
LIN {X 90.917,Y 36.115,Z 70.500,A 180.000,B 0.000,C 180.000} C_DIS
LIN {X 90.818,Y 36.036,Z 70.500,A 180.000,B 0.000,C 180.000} C_DIS
LIN {X 90.677,Y 35.936,Z 70.500,A 180.000,B 0.000,C 180.000} C_DIS
LIN {X 90.640,Y 35.912,Z 70.500,A 180.000,B 0.000,C 180.000} C_DIS
LIN {X 90.461,Y 35.809,Z 70.500,A 180.000,B 0.000,C 180.000} C_DIS
LIN {X 90.356,Y 35.757,Z 70.500,A 180.000,B 0.000,C 180.000} C_DIS
LIN {X 90.282,Y 35.724,Z 70.500,A 180.000,B 0.000,C 180.000} C_DIS
LIN {X 90.103,Y 35.656,Z 70.500,A 180.000,B 0.000,C 180.000} C_DIS
LIN {X 89.925,Y 35.603,Z 70.500,A 180.000,B 0.000,C 180.000} C_DIS
LIN {X 89.819,Y 35.578,Z 70.500,A 180.000,B 0.000,C 180.000} C_DIS
LIN {X 89.746,Y 35.564,Z 70.500,A 180.000,B 0.000,C 180.000} C_DIS
LIN {X 89.567,Y 35.539,Z 70.500,A 180.000,B 0.000,C 180.000} C_DIS
LIN {X 89.388,Y 35.526,Z 70.500,A 180.000,B 0.000,C 180.000} C_DIS
LIN {X 89.209,Y 35.526,Z 70.500,A 180.000,B 0.000,C 180.000} C_DIS
LIN {X 89.031,Y 35.540,Z 70.500,A 180.000,B 0.000,C 180.000} C_DIS
LIN {X 88.852,Y 35.566,Z 70.500,A 180.000,B 0.000,C 180.000} C_DIS
LIN {X 88.788,Y 35.578,Z 70.500,A 180.000,B 0.000,C 180.000} C_DIS
LIN {X 88.673,Y 35.605,Z 70.500,A 180.000,B 0.000,C 180.000} C_DIS
LIN {X 88.494,Y 35.659,Z 70.500,A 180.000,B 0.000,C 180.000} C_DIS
LIN {X 77.947,Y 39.217,Z 70.500,A 180.000,B 0.000,C 180.000} C_DIS
LIN {X 77.858,Y 39.248,Z 70.500,A 180.000,B 0.000,C 180.000} C_DIS
LIN {X 77.813,Y 39.263,Z 70.500,A 180.000,B 0.000,C 180.000} C_DIS
LIN {X 77.768,Y 39.280,Z 70.500,A 180.000,B 0.000,C 180.000} C_DIS
LIN {X 77.736,Y 39.292,Z 70.500,A 180.000,B 0.000,C 180.000} C_DIS
LIN {X 77.704,Y 39.305,Z 70.500,A 180.000,B 0.000,C 180.000} C_DIS
LIN {X 77.673,Y 39.319,Z 70.500,A 180.000,B 0.000,C 180.000} C_DIS
LIN {X 77.641,Y 39.333,Z 70.500,A 180.000,B 0.000,C 180.000} C_DIS
LIN {X 77.589,Y 39.356,Z 70.500,A 180.000,B 0.000,C 180.000} C_DIS
LIN {X 77.545,Y 39.378,Z 70.500,A 180.000,B 0.000,C 180.000} C_DIS
LIN {X 77.500,Y 39.401,Z 70.500,A 180.000,B 0.000,C 180.000} C_DIS
LIN {X 77.455,Y 39.425,Z 70.500,A 180.000,B 0.000,C 180.000} C_DIS
LIN {X 77.411,Y 39.450,Z 70.500,A 180.000,B 0.000,C 180.000} C_DIS
LIN {X 77.360,Y 39.480,Z 70.500,A 180.000,B 0.000,C 180.000} C_DIS
LIN {X 77.310,Y 39.511,Z 70.500,A 180.000,B 0.000,C 180.000} C_DIS
LIN {X 77.232,Y 39.564,Z 70.500,A 180.000,B 0.000,C 180.000} C_DIS
LIN {X 77.149,Y 39.624,Z 70.500,A 180.000,B 0.000,C 180.000} C_DIS
LIN {X 77.066,Y 39.690,Z 70.500,A 180.000,B 0.000,C 180.000} C_DIS
LIN {X 77.053,Y 39.701,Z 70.500,A 180.000,B 0.000,C 180.000} C_DIS
LIN {X 76.964,Y 39.780,Z 70.500,A 180.000,B 0.000,C 180.000} C_DIS
LIN {X 76.874,Y 39.867,Z 70.500,A 180.000,B 0.000,C 180.000} C_DIS
LIN {X 76.872,Y 39.869,Z 70.500,A 180.000,B 0.000,C 180.000} C_DIS
LIN {X 76.789,Y 39.958,Z 70.500,A 180.000,B 0.000,C 180.000} C_DIS
LIN {X 76.714,Y 40.048,Z 70.500,A 180.000,B 0.000,C 180.000} C_DIS
LIN {X 76.696,Y 40.070,Z 70.500,A 180.000,B 0.000,C 180.000} C_DIS
LIN {X 76.582,Y 40.226,Z 70.500,A 180.000,B 0.000,C 180.000} C_DIS
LIN {X 76.517,Y 40.330,Z 70.500,A 180.000,B 0.000,C 180.000} C_DIS
LIN {X 76.473,Y 40.405,Z 70.500,A 180.000,B 0.000,C 180.000} C_DIS
LIN {X 76.384,Y 40.584,Z 70.500,A 180.000,B 0.000,C 180.000} C_DIS
LIN {X 76.338,Y 40.692,Z 70.500,A 180.000,B 0.000,C 180.000} C_DIS
LIN {X 76.311,Y 40.763,Z 70.500,A 180.000,B 0.000,C 180.000} C_DIS
LIN {X 76.254,Y 40.942,Z 70.500,A 180.000,B 0.000,C 180.000} C_DIS
LIN {X 76.211,Y 41.120,Z 70.500,A 180.000,B 0.000,C 180.000} C_DIS
LIN {X 76.181,Y 41.299,Z 70.500,A 180.000,B 0.000,C 180.000} C_DIS
LIN {X 76.165,Y 41.478,Z 70.500,A 180.000,B 0.000,C 180.000} C_DIS
LIN {X 76.162,Y 41.657,Z 70.500,A 180.000,B 0.000,C 180.000} C_DIS
LIN {X 76.171,Y 41.835,Z 70.500,A 180.000,B 0.000,C 180.000} C_DIS
LIN {X 76.194,Y 42.014,Z 70.500,A 180.000,B 0.000,C 180.000} C_DIS
LIN {X 76.229,Y 42.193,Z 70.500,A 180.000,B 0.000,C 180.000} C_DIS
LIN {X 76.279,Y 42.372,Z 70.500,A 180.000,B 0.000,C 180.000} C_DIS
LIN {X 76.339,Y 42.550,Z 70.500,A 180.000,B 0.000,C 180.000} C_DIS
LIN {X 79.664,Y 52.406,Z 70.500,A 180.000,B 0.000,C 180.000} C_DIS
LIN {X 82.671,Y 61.321,Z 70.500,A 180.000,B 0.000,C 180.000} C_DIS
LIN {X 82.736,Y 61.500,Z 70.500,A 180.000,B 0.000,C 180.000} C_DIS
LIN {X 82.774,Y 61.589,Z 70.500,A 180.000,B 0.000,C 180.000} C_DIS
LIN {X 82.816,Y 61.679,Z 70.500,A 180.000,B 0.000,C 180.000} C_DIS
LIN {X 82.914,Y 61.858,Z 70.500,A 180.000,B 0.000,C 180.000} C_DIS
LIN {X 82.952,Y 61.919,Z 70.500,A 180.000,B 0.000,C 180.000} C_DIS
LIN {X 83.033,Y 62.036,Z 70.500,A 180.000,B 0.000,C 180.000} C_DIS
LIN {X 83.131,Y 62.163,Z 70.500,A 180.000,B 0.000,C 180.000} C_DIS
LIN {X 83.176,Y 62.215,Z 70.500,A 180.000,B 0.000,C 180.000} C_DIS
LIN {X 83.310,Y 62.356,Z 70.500,A 180.000,B 0.000,C 180.000} C_DIS
LIN {X 83.350,Y 62.394,Z 70.500,A 180.000,B 0.000,C 180.000} C_DIS
LIN {X 83.489,Y 62.515,Z 70.500,A 180.000,B 0.000,C 180.000} C_DIS
LIN {X 83.564,Y 62.573,Z 70.500,A 180.000,B 0.000,C 180.000} C_DIS
LIN {X 83.668,Y 62.646,Z 70.500,A 180.000,B 0.000,C 180.000} C_DIS
LIN {X 83.841,Y 62.751,Z 70.500,A 180.000,B 0.000,C 180.000} C_DIS
LIN {X 83.846,Y 62.754,Z 70.500,A 180.000,B 0.000,C 180.000} C_DIS
LIN {X 84.025,Y 62.844,Z 70.500,A 180.000,B 0.000,C 180.000} C_DIS
LIN {X 84.204,Y 62.916,Z 70.500,A 180.000,B 0.000,C 180.000} C_DIS
LIN {X 84.243,Y 62.930,Z 70.500,A 180.000,B 0.000,C 180.000} C_DIS
LIN {X 84.383,Y 62.974,Z 70.500,A 180.000,B 0.000,C 180.000} C_DIS
LIN {X 84.561,Y 63.016,Z 70.500,A 180.000,B 0.000,C 180.000} C_DIS
LIN {X 84.740,Y 63.046,Z 70.500,A 180.000,B 0.000,C 180.000} C_DIS
LIN {X 84.830,Y 63.055,Z 70.500,A 180.000,B 0.000,C 180.000} C_DIS
LIN {X 84.919,Y 63.062,Z 70.500,A 180.000,B 0.000,C 180.000} C_DIS
LIN {X 85.008,Y 63.065,Z 70.500,A 180.000,B 0.000,C 180.000} C_DIS
LIN {X 85.098,Y 63.065,Z 70.500,A 180.000,B 0.000,C 180.000} C_DIS
LIN {X 85.187,Y 63.062,Z 70.500,A 180.000,B 0.000,C 180.000} C_DIS
LIN {X 85.276,Y 63.056,Z 70.500,A 180.000,B 0.000,C 180.000} C_DIS
LIN {X 85.366,Y 63.046,Z 70.500,A 180.000,B 0.000,C 180.000} C_DIS
LIN {X 85.411,Y 63.040,Z 70.500,A 180.000,B 0.000,C 180.000} C_DIS
LIN {X 85.455,Y 63.033,Z 70.500,A 180.000,B 0.000,C 180.000} C_DIS
LIN {X 85.500,Y 63.025,Z 70.500,A 180.000,B 0.000,C 180.000} C_DIS
LIN {X 85.545,Y 63.017,Z 70.500,A 180.000,B 0.000,C 180.000} C_DIS
LIN {X 85.589,Y 63.008,Z 70.500,A 180.000,B 0.000,C 180.000} C_DIS
LIN {X 85.634,Y 62.997,Z 70.500,A 180.000,B 0.000,C 180.000} C_DIS
LIN {X 85.679,Y 62.986,Z 70.500,A 180.000,B 0.000,C 180.000} C_DIS
LIN {X 85.723,Y 62.974,Z 70.500,A 180.000,B 0.000,C 180.000} C_DIS
LIN {X 85.768,Y 62.961,Z 70.500,A 180.000,B 0.000,C 180.000} C_DIS
LIN {X 85.813,Y 62.948,Z 70.500,A 180.000,B 0.000,C 180.000} C_DIS
LIN {X 85.866,Y 62.930,Z 70.500,A 180.000,B 0.000,C 180.000} C_DIS
LIN {X 96.464,Y 59.355,Z 70.500,A 180.000,B 0.000,C 180.000} C_DIS
LIN {X 96.539,Y 59.329,Z 70.500,A 180.000,B 0.000,C 180.000} C_DIS
LIN {X 96.718,Y 59.257,Z 70.500,A 180.000,B 0.000,C 180.000} C_DIS
LIN {X 96.883,Y 59.176,Z 70.500,A 180.000,B 0.000,C 180.000} C_DIS
LIN {X 96.897,Y 59.169,Z 70.500,A 180.000,B 0.000,C 180.000} C_DIS
LIN {X 97.075,Y 59.061,Z 70.500,A 180.000,B 0.000,C 180.000} C_DIS
LIN {X 97.167,Y 58.997,Z 70.500,A 180.000,B 0.000,C 180.000} C_DIS
LIN {X 97.254,Y 58.931,Z 70.500,A 180.000,B 0.000,C 180.000} C_DIS
LIN {X 97.385,Y 58.819,Z 70.500,A 180.000,B 0.000,C 180.000} C_DIS
LIN {X 97.433,Y 58.774,Z 70.500,A 180.000,B 0.000,C 180.000} C_DIS
LIN {X 97.562,Y 58.640,Z 70.500,A 180.000,B 0.000,C 180.000} C_DIS
LIN {X 97.612,Y 58.582,Z 70.500,A 180.000,B 0.000,C 180.000} C_DIS
LIN {X 97.707,Y 58.461,Z 70.500,A 180.000,B 0.000,C 180.000} C_DIS
LIN {X 97.790,Y 58.341,Z 70.500,A 180.000,B 0.000,C 180.000} C_DIS
LIN {X 97.828,Y 58.282,Z 70.500,A 180.000,B 0.000,C 180.000} C_DIS
LIN {X 97.928,Y 58.103,Z 70.500,A 180.000,B 0.000,C 180.000} C_DIS
LIN {X 97.969,Y 58.017,Z 70.500,A 180.000,B 0.000,C 180.000} C_DIS
LIN {X 98.009,Y 57.925,Z 70.500,A 180.000,B 0.000,C 180.000} C_DIS
LIN {X 98.075,Y 57.746,Z 70.500,A 180.000,B 0.000,C 180.000} C_DIS
LIN {X 98.125,Y 57.567,Z 70.500,A 180.000,B 0.000,C 180.000} C_DIS
LIN {X 98.148,Y 57.466,Z 70.500,A 180.000,B 0.000,C 180.000} C_DIS
LIN {X 98.162,Y 57.388,Z 70.500,A 180.000,B 0.000,C 180.000} C_DIS
LIN {X 98.186,Y 57.210,Z 70.500,A 180.000,B 0.000,C 180.000} C_DIS
LIN {X 98.196,Y 57.031,Z 70.500,A 180.000,B 0.000,C 180.000} C_DIS
LIN {X 98.193,Y 56.852,Z 70.500,A 180.000,B 0.000,C 180.000} C_DIS
LIN {X 98.178,Y 56.673,Z 70.500,A 180.000,B 0.000,C 180.000} C_DIS
LIN {X 98.150,Y 56.495,Z 70.500,A 180.000,B 0.000,C 180.000} C_DIS
LIN {X 98.148,Y 56.485,Z 70.500,A 180.000,B 0.000,C 180.000} C_DIS
LIN {X 98.108,Y 56.316,Z 70.500,A 180.000,B 0.000,C 180.000} C_DIS
LIN {X 98.052,Y 56.137,Z 70.500,A 180.000,B 0.000,C 180.000} C_DIS
LIN {X 94.699,Y 46.199,Z 70.500,A 180.000,B 0.000,C 180.000} C_DIS
; Lead Out Move Starts
LIN {X 94.770,Y 45.743,Z 70.500,A 180.000,B 0.000,C 180.000} C_DIS
LIN {X 95.184,Y 45.539,Z 70.500,A 180.000,B 0.000,C 180.000} C_DIS
LIN {X 95.900,Y 45.554,Z 70.500,A 180.000,B 0.000,C 180.000} C_DIS
LIN {X 96.253,Y 45.561,Z 70.646,A 180.000,B 0.000,C 180.000} C_DIS
LIN {X 96.400,Y 45.565,Z 71.000,A 180.000,B 0.000,C 180.000} C_DIS
; Rapid Move Starts
LIN {X 96.400,Y 45.565,Z 95.000,A 180.000,B 0.000,C 180.000} C_DIS
LIN {X 78.807,Y 51.609,Z 95.000,A 180.000,B 0.000,C 180.000} C_DIS
LIN {X 78.807,Y 51.609,Z 72.598,A 180.000,B 0.000,C 180.000} C_DIS
; Plunge Move Starts
$VEL.CP=0.01
LIN {X 78.807,Y 51.609,Z 71.625,A 180.000,B 0.000,C 180.000} C_DIS
; Lead In Move Starts
LIN {X 78.807,Y 51.609,Z 70.500,A 180.000,B 0.000,C 180.000} C_DIS
LIN {X 78.748,Y 51.580,Z 70.500,A 180.000,B 0.000,C 180.000} C_DIS
; Cutting Move Starts
$VEL.CP=0.02
LIN {X 75.762,Y 42.729,Z 70.500,A 180.000,B 0.000,C 180.000} C_DIS
LIN {X 75.701,Y 42.550,Z 70.500,A 180.000,B 0.000,C 180.000} C_DIS
LIN {X 75.628,Y 42.372,Z 70.500,A 180.000,B 0.000,C 180.000} C_DIS
LIN {X 75.623,Y 42.361,Z 70.500,A 180.000,B 0.000,C 180.000} C_DIS
LIN {X 75.538,Y 42.193,Z 70.500,A 180.000,B 0.000,C 180.000} C_DIS
LIN {X 75.444,Y 42.038,Z 70.500,A 180.000,B 0.000,C 180.000} C_DIS
LIN {X 75.429,Y 42.014,Z 70.500,A 180.000,B 0.000,C 180.000} C_DIS
LIN {X 75.297,Y 41.835,Z 70.500,A 180.000,B 0.000,C 180.000} C_DIS
LIN {X 75.265,Y 41.797,Z 70.500,A 180.000,B 0.000,C 180.000} C_DIS
LIN {X 75.138,Y 41.657,Z 70.500,A 180.000,B 0.000,C 180.000} C_DIS
LIN {X 75.087,Y 41.606,Z 70.500,A 180.000,B 0.000,C 180.000} C_DIS
LIN {X 74.943,Y 41.478,Z 70.500,A 180.000,B 0.000,C 180.000} C_DIS
LIN {X 74.908,Y 41.449,Z 70.500,A 180.000,B 0.000,C 180.000} C_DIS
LIN {X 74.729,Y 41.319,Z 70.500,A 180.000,B 0.000,C 180.000} C_DIS
LIN {X 74.698,Y 41.299,Z 70.500,A 180.000,B 0.000,C 180.000} C_DIS
LIN {X 74.550,Y 41.212,Z 70.500,A 180.000,B 0.000,C 180.000} C_DIS
LIN {X 74.372,Y 41.123,Z 70.500,A 180.000,B 0.000,C 180.000} C_DIS
LIN {X 74.365,Y 41.120,Z 70.500,A 180.000,B 0.000,C 180.000} C_DIS
LIN {X 74.193,Y 41.052,Z 70.500,A 180.000,B 0.000,C 180.000} C_DIS
LIN {X 74.014,Y 40.995,Z 70.500,A 180.000,B 0.000,C 180.000} C_DIS
LIN {X 73.835,Y 40.953,Z 70.500,A 180.000,B 0.000,C 180.000} C_DIS
LIN {X 73.772,Y 40.942,Z 70.500,A 180.000,B 0.000,C 180.000} C_DIS
LIN {X 73.656,Y 40.925,Z 70.500,A 180.000,B 0.000,C 180.000} C_DIS
LIN {X 73.567,Y 40.915,Z 70.500,A 180.000,B 0.000,C 180.000} C_DIS
LIN {X 73.478,Y 40.909,Z 70.500,A 180.000,B 0.000,C 180.000} C_DIS
LIN {X 73.388,Y 40.906,Z 70.500,A 180.000,B 0.000,C 180.000} C_DIS
LIN {X 73.299,Y 40.906,Z 70.500,A 180.000,B 0.000,C 180.000} C_DIS
LIN {X 73.210,Y 40.910,Z 70.500,A 180.000,B 0.000,C 180.000} C_DIS
LIN {X 73.120,Y 40.917,Z 70.500,A 180.000,B 0.000,C 180.000} C_DIS
LIN {X 73.031,Y 40.927,Z 70.500,A 180.000,B 0.000,C 180.000} C_DIS
LIN {X 72.986,Y 40.933,Z 70.500,A 180.000,B 0.000,C 180.000} C_DIS
LIN {X 72.941,Y 40.940,Z 70.500,A 180.000,B 0.000,C 180.000} C_DIS
LIN {X 72.931,Y 40.942,Z 70.500,A 180.000,B 0.000,C 180.000} C_DIS
LIN {X 72.889,Y 40.949,Z 70.500,A 180.000,B 0.000,C 180.000} C_DIS
LIN {X 72.847,Y 40.957,Z 70.500,A 180.000,B 0.000,C 180.000} C_DIS
LIN {X 72.805,Y 40.967,Z 70.500,A 180.000,B 0.000,C 180.000} C_DIS
LIN {X 72.763,Y 40.976,Z 70.500,A 180.000,B 0.000,C 180.000} C_DIS
LIN {X 72.718,Y 40.988,Z 70.500,A 180.000,B 0.000,C 180.000} C_DIS
LIN {X 72.673,Y 41.000,Z 70.500,A 180.000,B 0.000,C 180.000} C_DIS
LIN {X 72.629,Y 41.013,Z 70.500,A 180.000,B 0.000,C 180.000} C_DIS
LIN {X 72.584,Y 41.027,Z 70.500,A 180.000,B 0.000,C 180.000} C_DIS
LIN {X 72.405,Y 41.087,Z 70.500,A 180.000,B 0.000,C 180.000} C_DIS
LIN {X 45.590,Y 50.133,Z 70.500,A 180.000,B 0.000,C 180.000} C_DIS
LIN {X 45.411,Y 50.194,Z 70.500,A 180.000,B 0.000,C 180.000} C_DIS
LIN {X 45.296,Y 50.238,Z 70.500,A 180.000,B 0.000,C 180.000} C_DIS
LIN {X 45.232,Y 50.265,Z 70.500,A 180.000,B 0.000,C 180.000} C_DIS
LIN {X 45.053,Y 50.353,Z 70.500,A 180.000,B 0.000,C 180.000} C_DIS
LIN {X 44.944,Y 50.416,Z 70.500,A 180.000,B 0.000,C 180.000} C_DIS
LIN {X 44.874,Y 50.461,Z 70.500,A 180.000,B 0.000,C 180.000} C_DIS
LIN {X 44.785,Y 50.522,Z 70.500,A 180.000,B 0.000,C 180.000} C_DIS
LIN {X 44.696,Y 50.590,Z 70.500,A 180.000,B 0.000,C 180.000} C_DIS
LIN {X 44.689,Y 50.595,Z 70.500,A 180.000,B 0.000,C 180.000} C_DIS
LIN {X 44.603,Y 50.667,Z 70.500,A 180.000,B 0.000,C 180.000} C_DIS
LIN {X 44.517,Y 50.746,Z 70.500,A 180.000,B 0.000,C 180.000} C_DIS
LIN {X 44.488,Y 50.774,Z 70.500,A 180.000,B 0.000,C 180.000} C_DIS
LIN {X 44.410,Y 50.855,Z 70.500,A 180.000,B 0.000,C 180.000} C_DIS
LIN {X 44.338,Y 50.936,Z 70.500,A 180.000,B 0.000,C 180.000} C_DIS
LIN {X 44.325,Y 50.953,Z 70.500,A 180.000,B 0.000,C 180.000} C_DIS
LIN {X 44.254,Y 51.042,Z 70.500,A 180.000,B 0.000,C 180.000} C_DIS
LIN {X 44.189,Y 51.131,Z 70.500,A 180.000,B 0.000,C 180.000} C_DIS
LIN {X 44.159,Y 51.176,Z 70.500,A 180.000,B 0.000,C 180.000} C_DIS
LIN {X 44.077,Y 51.310,Z 70.500,A 180.000,B 0.000,C 180.000} C_DIS
LIN {X 43.984,Y 51.489,Z 70.500,A 180.000,B 0.000,C 180.000} C_DIS
LIN {X 43.981,Y 51.497,Z 70.500,A 180.000,B 0.000,C 180.000} C_DIS
LIN {X 43.909,Y 51.668,Z 70.500,A 180.000,B 0.000,C 180.000} C_DIS
LIN {X 43.849,Y 51.847,Z 70.500,A 180.000,B 0.000,C 180.000} C_DIS
LIN {X 43.804,Y 52.025,Z 70.500,A 180.000,B 0.000,C 180.000} C_DIS
LIN {X 43.802,Y 52.035,Z 70.500,A 180.000,B 0.000,C 180.000} C_DIS
LIN {X 43.772,Y 52.204,Z 70.500,A 180.000,B 0.000,C 180.000} C_DIS
LIN {X 43.754,Y 52.383,Z 70.500,A 180.000,B 0.000,C 180.000} C_DIS
LIN {X 43.748,Y 52.562,Z 70.500,A 180.000,B 0.000,C 180.000} C_DIS
LIN {X 43.756,Y 52.740,Z 70.500,A 180.000,B 0.000,C 180.000} C_DIS
LIN {X 43.776,Y 52.919,Z 70.500,A 180.000,B 0.000,C 180.000} C_DIS
LIN {X 43.802,Y 53.064,Z 70.500,A 180.000,B 0.000,C 180.000} C_DIS
LIN {X 43.809,Y 53.098,Z 70.500,A 180.000,B 0.000,C 180.000} C_DIS
LIN {X 43.856,Y 53.277,Z 70.500,A 180.000,B 0.000,C 180.000} C_DIS
LIN {X 43.916,Y 53.455,Z 70.500,A 180.000,B 0.000,C 180.000} C_DIS
LIN {X 50.248,Y 72.226,Z 70.500,A 180.000,B 0.000,C 180.000} C_DIS
LIN {X 50.311,Y 72.405,Z 70.500,A 180.000,B 0.000,C 180.000} C_DIS
LIN {X 50.388,Y 72.584,Z 70.500,A 180.000,B 0.000,C 180.000} C_DIS
LIN {X 50.416,Y 72.640,Z 70.500,A 180.000,B 0.000,C 180.000} C_DIS
LIN {X 50.484,Y 72.763,Z 70.500,A 180.000,B 0.000,C 180.000} C_DIS
LIN {X 50.595,Y 72.936,Z 70.500,A 180.000,B 0.000,C 180.000} C_DIS
LIN {X 50.599,Y 72.941,Z 70.500,A 180.000,B 0.000,C 180.000} C_DIS
LIN {X 50.665,Y 73.031,Z 70.500,A 180.000,B 0.000,C 180.000} C_DIS
LIN {X 50.737,Y 73.120,Z 70.500,A 180.000,B 0.000,C 180.000} C_DIS
LIN {X 50.774,Y 73.162,Z 70.500,A 180.000,B 0.000,C 180.000} C_DIS
LIN {X 50.905,Y 73.299,Z 70.500,A 180.000,B 0.000,C 180.000} C_DIS
LIN {X 50.953,Y 73.343,Z 70.500,A 180.000,B 0.000,C 180.000} C_DIS
LIN {X 51.112,Y 73.478,Z 70.500,A 180.000,B 0.000,C 180.000} C_DIS
LIN {X 51.131,Y 73.493,Z 70.500,A 180.000,B 0.000,C 180.000} C_DIS
LIN {X 51.310,Y 73.616,Z 70.500,A 180.000,B 0.000,C 180.000} C_DIS
LIN {X 51.376,Y 73.656,Z 70.500,A 180.000,B 0.000,C 180.000} C_DIS
LIN {X 51.489,Y 73.719,Z 70.500,A 180.000,B 0.000,C 180.000} C_DIS
LIN {X 51.668,Y 73.803,Z 70.500,A 180.000,B 0.000,C 180.000} C_DIS
LIN {X 51.749,Y 73.835,Z 70.500,A 180.000,B 0.000,C 180.000} C_DIS
LIN {X 51.847,Y 73.870,Z 70.500,A 180.000,B 0.000,C 180.000} C_DIS
LIN {X 52.025,Y 73.923,Z 70.500,A 180.000,B 0.000,C 180.000} C_DIS
LIN {X 52.204,Y 73.961,Z 70.500,A 180.000,B 0.000,C 180.000} C_DIS
LIN {X 52.383,Y 73.987,Z 70.500,A 180.000,B 0.000,C 180.000} C_DIS
LIN {X 52.562,Y 73.999,Z 70.500,A 180.000,B 0.000,C 180.000} C_DIS
LIN {X 52.740,Y 73.998,Z 70.500,A 180.000,B 0.000,C 180.000} C_DIS
LIN {X 52.919,Y 73.985,Z 70.500,A 180.000,B 0.000,C 180.000} C_DIS
LIN {X 53.098,Y 73.958,Z 70.500,A 180.000,B 0.000,C 180.000} C_DIS
LIN {X 53.277,Y 73.918,Z 70.500,A 180.000,B 0.000,C 180.000} C_DIS
LIN {X 53.455,Y 73.864,Z 70.500,A 180.000,B 0.000,C 180.000} C_DIS
LIN {X 80.450,Y 64.757,Z 70.500,A 180.000,B 0.000,C 180.000} C_DIS
LIN {X 80.566,Y 64.718,Z 70.500,A 180.000,B 0.000,C 180.000} C_DIS
LIN {X 80.628,Y 64.695,Z 70.500,A 180.000,B 0.000,C 180.000} C_DIS
LIN {X 80.673,Y 64.678,Z 70.500,A 180.000,B 0.000,C 180.000} C_DIS
LIN {X 80.718,Y 64.660,Z 70.500,A 180.000,B 0.000,C 180.000} C_DIS
LIN {X 80.763,Y 64.640,Z 70.500,A 180.000,B 0.000,C 180.000} C_DIS
LIN {X 80.807,Y 64.620,Z 70.500,A 180.000,B 0.000,C 180.000} C_DIS
LIN {X 80.846,Y 64.601,Z 70.500,A 180.000,B 0.000,C 180.000} C_DIS
LIN {X 80.886,Y 64.581,Z 70.500,A 180.000,B 0.000,C 180.000} C_DIS
LIN {X 80.925,Y 64.561,Z 70.500,A 180.000,B 0.000,C 180.000} C_DIS
LIN {X 80.964,Y 64.539,Z 70.500,A 180.000,B 0.000,C 180.000} C_DIS
LIN {X 80.986,Y 64.527,Z 70.500,A 180.000,B 0.000,C 180.000} C_DIS
LIN {X 81.031,Y 64.501,Z 70.500,A 180.000,B 0.000,C 180.000} C_DIS
LIN {X 81.075,Y 64.473,Z 70.500,A 180.000,B 0.000,C 180.000} C_DIS
LIN {X 81.165,Y 64.414,Z 70.500,A 180.000,B 0.000,C 180.000} C_DIS
LIN {X 81.240,Y 64.360,Z 70.500,A 180.000,B 0.000,C 180.000} C_DIS
LIN {X 81.344,Y 64.279,Z 70.500,A 180.000,B 0.000,C 180.000} C_DIS
LIN {X 81.453,Y 64.182,Z 70.500,A 180.000,B 0.000,C 180.000} C_DIS
LIN {X 81.522,Y 64.115,Z 70.500,A 180.000,B 0.000,C 180.000} C_DIS
LIN {X 81.626,Y 64.003,Z 70.500,A 180.000,B 0.000,C 180.000} C_DIS
LIN {X 81.701,Y 63.913,Z 70.500,A 180.000,B 0.000,C 180.000} C_DIS
LIN {X 81.769,Y 63.824,Z 70.500,A 180.000,B 0.000,C 180.000} C_DIS
LIN {X 81.880,Y 63.657,Z 70.500,A 180.000,B 0.000,C 180.000} C_DIS
LIN {X 81.887,Y 63.645,Z 70.500,A 180.000,B 0.000,C 180.000} C_DIS
LIN {X 81.985,Y 63.467,Z 70.500,A 180.000,B 0.000,C 180.000} C_DIS
LIN {X 82.059,Y 63.303,Z 70.500,A 180.000,B 0.000,C 180.000} C_DIS
LIN {X 82.065,Y 63.288,Z 70.500,A 180.000,B 0.000,C 180.000} C_DIS
LIN {X 82.129,Y 63.109,Z 70.500,A 180.000,B 0.000,C 180.000} C_DIS
LIN {X 82.178,Y 62.930,Z 70.500,A 180.000,B 0.000,C 180.000} C_DIS
LIN {X 82.213,Y 62.751,Z 70.500,A 180.000,B 0.000,C 180.000} C_DIS
LIN {X 82.236,Y 62.573,Z 70.500,A 180.000,B 0.000,C 180.000} C_DIS
LIN {X 82.237,Y 62.550,Z 70.500,A 180.000,B 0.000,C 180.000} C_DIS
LIN {X 82.245,Y 62.394,Z 70.500,A 180.000,B 0.000,C 180.000} C_DIS
LIN {X 82.241,Y 62.215,Z 70.500,A 180.000,B 0.000,C 180.000} C_DIS
LIN {X 82.237,Y 62.164,Z 70.500,A 180.000,B 0.000,C 180.000} C_DIS
LIN {X 82.224,Y 62.036,Z 70.500,A 180.000,B 0.000,C 180.000} C_DIS
LIN {X 82.195,Y 61.858,Z 70.500,A 180.000,B 0.000,C 180.000} C_DIS
LIN {X 82.151,Y 61.679,Z 70.500,A 180.000,B 0.000,C 180.000} C_DIS
LIN {X 82.094,Y 61.500,Z 70.500,A 180.000,B 0.000,C 180.000} C_DIS
LIN {X 78.748,Y 51.580,Z 70.500,A 180.000,B 0.000,C 180.000} C_DIS
; Lead Out Move Starts
LIN {X 78.777,Y 51.521,Z 70.500,A 180.000,B 0.000,C 180.000} C_DIS
; Rapid Move Starts
LIN {X 78.777,Y 51.521,Z 95.000,A 180.000,B 0.000,C 180.000} C_DIS
LIN {X 75.266,Y 40.718,Z 95.000,A 180.000,B 0.000,C 180.000} C_DIS
LIN {X 75.266,Y 40.718,Z 72.339,A 180.000,B 0.000,C 180.000} C_DIS
; Plunge Move Starts
$VEL.CP=0.01
LIN {X 75.266,Y 40.718,Z 71.372,A 180.000,B 0.000,C 180.000} C_DIS
; Lead In Move Starts
LIN {X 75.266,Y 40.718,Z 70.247,A 180.000,B 0.000,C 180.000} C_DIS
LIN {X 75.184,Y 40.763,Z 70.247,A 180.000,B 0.000,C 180.000} C_DIS
; Cutting Move Starts
$VEL.CP=0.02
LIN {X 75.087,Y 40.727,Z 70.247,A 180.000,B 0.000,C 180.000} C_DIS
LIN {X 74.908,Y 40.674,Z 70.247,A 180.000,B 0.000,C 180.000} C_DIS
LIN {X 74.729,Y 40.634,Z 70.247,A 180.000,B 0.000,C 180.000} C_DIS
LIN {X 74.550,Y 40.608,Z 70.247,A 180.000,B 0.000,C 180.000} C_DIS
LIN {X 74.372,Y 40.595,Z 70.247,A 180.000,B 0.000,C 180.000} C_DIS
LIN {X 74.282,Y 40.593,Z 70.247,A 180.000,B 0.000,C 180.000} C_DIS
LIN {X 74.193,Y 40.595,Z 70.247,A 180.000,B 0.000,C 180.000} C_DIS
LIN {X 74.103,Y 40.599,Z 70.247,A 180.000,B 0.000,C 180.000} C_DIS
LIN {X 74.014,Y 40.607,Z 70.247,A 180.000,B 0.000,C 180.000} C_DIS
LIN {X 73.969,Y 40.612,Z 70.247,A 180.000,B 0.000,C 180.000} C_DIS
LIN {X 73.925,Y 40.618,Z 70.247,A 180.000,B 0.000,C 180.000} C_DIS
LIN {X 73.880,Y 40.625,Z 70.247,A 180.000,B 0.000,C 180.000} C_DIS
LIN {X 73.835,Y 40.633,Z 70.247,A 180.000,B 0.000,C 180.000} C_DIS
LIN {X 73.791,Y 40.641,Z 70.247,A 180.000,B 0.000,C 180.000} C_DIS
LIN {X 73.746,Y 40.651,Z 70.247,A 180.000,B 0.000,C 180.000} C_DIS
LIN {X 73.701,Y 40.661,Z 70.247,A 180.000,B 0.000,C 180.000} C_DIS
LIN {X 73.656,Y 40.672,Z 70.247,A 180.000,B 0.000,C 180.000} C_DIS
LIN {X 73.634,Y 40.678,Z 70.247,A 180.000,B 0.000,C 180.000} C_DIS
LIN {X 73.612,Y 40.684,Z 70.247,A 180.000,B 0.000,C 180.000} C_DIS
LIN {X 73.589,Y 40.690,Z 70.247,A 180.000,B 0.000,C 180.000} C_DIS
LIN {X 73.567,Y 40.697,Z 70.247,A 180.000,B 0.000,C 180.000} C_DIS
LIN {X 73.545,Y 40.703,Z 70.247,A 180.000,B 0.000,C 180.000} C_DIS
LIN {X 73.522,Y 40.710,Z 70.247,A 180.000,B 0.000,C 180.000} C_DIS
LIN {X 73.500,Y 40.718,Z 70.247,A 180.000,B 0.000,C 180.000} C_DIS
LIN {X 73.478,Y 40.725,Z 70.247,A 180.000,B 0.000,C 180.000} C_DIS
LIN {X 45.590,Y 50.133,Z 70.247,A 180.000,B 0.000,C 180.000} C_DIS
LIN {X 45.411,Y 50.194,Z 70.247,A 180.000,B 0.000,C 180.000} C_DIS
LIN {X 45.296,Y 50.238,Z 70.247,A 180.000,B 0.000,C 180.000} C_DIS
LIN {X 45.232,Y 50.265,Z 70.247,A 180.000,B 0.000,C 180.000} C_DIS
LIN {X 45.053,Y 50.353,Z 70.247,A 180.000,B 0.000,C 180.000} C_DIS
LIN {X 44.944,Y 50.416,Z 70.247,A 180.000,B 0.000,C 180.000} C_DIS
LIN {X 44.874,Y 50.461,Z 70.247,A 180.000,B 0.000,C 180.000} C_DIS
LIN {X 44.785,Y 50.522,Z 70.247,A 180.000,B 0.000,C 180.000} C_DIS
LIN {X 44.696,Y 50.590,Z 70.247,A 180.000,B 0.000,C 180.000} C_DIS
LIN {X 44.689,Y 50.595,Z 70.247,A 180.000,B 0.000,C 180.000} C_DIS
LIN {X 44.603,Y 50.667,Z 70.247,A 180.000,B 0.000,C 180.000} C_DIS
LIN {X 44.517,Y 50.746,Z 70.247,A 180.000,B 0.000,C 180.000} C_DIS
LIN {X 44.488,Y 50.774,Z 70.247,A 180.000,B 0.000,C 180.000} C_DIS
LIN {X 44.410,Y 50.855,Z 70.247,A 180.000,B 0.000,C 180.000} C_DIS
LIN {X 44.338,Y 50.936,Z 70.247,A 180.000,B 0.000,C 180.000} C_DIS
LIN {X 44.325,Y 50.953,Z 70.247,A 180.000,B 0.000,C 180.000} C_DIS
LIN {X 44.254,Y 51.042,Z 70.247,A 180.000,B 0.000,C 180.000} C_DIS
LIN {X 44.189,Y 51.131,Z 70.247,A 180.000,B 0.000,C 180.000} C_DIS
LIN {X 44.159,Y 51.176,Z 70.247,A 180.000,B 0.000,C 180.000} C_DIS
LIN {X 44.077,Y 51.310,Z 70.247,A 180.000,B 0.000,C 180.000} C_DIS
LIN {X 43.984,Y 51.489,Z 70.247,A 180.000,B 0.000,C 180.000} C_DIS
LIN {X 43.981,Y 51.497,Z 70.247,A 180.000,B 0.000,C 180.000} C_DIS
LIN {X 43.909,Y 51.668,Z 70.247,A 180.000,B 0.000,C 180.000} C_DIS
LIN {X 43.849,Y 51.847,Z 70.247,A 180.000,B 0.000,C 180.000} C_DIS
LIN {X 43.804,Y 52.025,Z 70.247,A 180.000,B 0.000,C 180.000} C_DIS
LIN {X 43.802,Y 52.035,Z 70.247,A 180.000,B 0.000,C 180.000} C_DIS
LIN {X 43.772,Y 52.204,Z 70.247,A 180.000,B 0.000,C 180.000} C_DIS
LIN {X 43.754,Y 52.383,Z 70.247,A 180.000,B 0.000,C 180.000} C_DIS
LIN {X 43.748,Y 52.562,Z 70.247,A 180.000,B 0.000,C 180.000} C_DIS
LIN {X 43.756,Y 52.740,Z 70.247,A 180.000,B 0.000,C 180.000} C_DIS
LIN {X 43.776,Y 52.919,Z 70.247,A 180.000,B 0.000,C 180.000} C_DIS
LIN {X 43.802,Y 53.064,Z 70.247,A 180.000,B 0.000,C 180.000} C_DIS
LIN {X 43.809,Y 53.098,Z 70.247,A 180.000,B 0.000,C 180.000} C_DIS
LIN {X 43.856,Y 53.277,Z 70.247,A 180.000,B 0.000,C 180.000} C_DIS
LIN {X 43.916,Y 53.455,Z 70.247,A 180.000,B 0.000,C 180.000} C_DIS
LIN {X 50.248,Y 72.226,Z 70.247,A 180.000,B 0.000,C 180.000} C_DIS
LIN {X 50.311,Y 72.405,Z 70.247,A 180.000,B 0.000,C 180.000} C_DIS
LIN {X 50.388,Y 72.584,Z 70.247,A 180.000,B 0.000,C 180.000} C_DIS
LIN {X 50.416,Y 72.640,Z 70.247,A 180.000,B 0.000,C 180.000} C_DIS
LIN {X 50.484,Y 72.763,Z 70.247,A 180.000,B 0.000,C 180.000} C_DIS
LIN {X 50.595,Y 72.936,Z 70.247,A 180.000,B 0.000,C 180.000} C_DIS
LIN {X 50.599,Y 72.941,Z 70.247,A 180.000,B 0.000,C 180.000} C_DIS
LIN {X 50.665,Y 73.031,Z 70.247,A 180.000,B 0.000,C 180.000} C_DIS
LIN {X 50.737,Y 73.120,Z 70.247,A 180.000,B 0.000,C 180.000} C_DIS
LIN {X 50.774,Y 73.162,Z 70.247,A 180.000,B 0.000,C 180.000} C_DIS
LIN {X 50.905,Y 73.299,Z 70.247,A 180.000,B 0.000,C 180.000} C_DIS
LIN {X 50.953,Y 73.343,Z 70.247,A 180.000,B 0.000,C 180.000} C_DIS
LIN {X 51.112,Y 73.478,Z 70.247,A 180.000,B 0.000,C 180.000} C_DIS
LIN {X 51.131,Y 73.493,Z 70.247,A 180.000,B 0.000,C 180.000} C_DIS
LIN {X 51.310,Y 73.616,Z 70.247,A 180.000,B 0.000,C 180.000} C_DIS
LIN {X 51.376,Y 73.656,Z 70.247,A 180.000,B 0.000,C 180.000} C_DIS
LIN {X 51.489,Y 73.719,Z 70.247,A 180.000,B 0.000,C 180.000} C_DIS
LIN {X 51.668,Y 73.803,Z 70.247,A 180.000,B 0.000,C 180.000} C_DIS
LIN {X 51.749,Y 73.835,Z 70.247,A 180.000,B 0.000,C 180.000} C_DIS
LIN {X 51.847,Y 73.870,Z 70.247,A 180.000,B 0.000,C 180.000} C_DIS
LIN {X 52.025,Y 73.923,Z 70.247,A 180.000,B 0.000,C 180.000} C_DIS
LIN {X 52.204,Y 73.961,Z 70.247,A 180.000,B 0.000,C 180.000} C_DIS
LIN {X 52.383,Y 73.987,Z 70.247,A 180.000,B 0.000,C 180.000} C_DIS
LIN {X 52.562,Y 73.999,Z 70.247,A 180.000,B 0.000,C 180.000} C_DIS
LIN {X 52.740,Y 73.998,Z 70.247,A 180.000,B 0.000,C 180.000} C_DIS
LIN {X 52.919,Y 73.985,Z 70.247,A 180.000,B 0.000,C 180.000} C_DIS
LIN {X 53.098,Y 73.958,Z 70.247,A 180.000,B 0.000,C 180.000} C_DIS
LIN {X 53.277,Y 73.918,Z 70.247,A 180.000,B 0.000,C 180.000} C_DIS
LIN {X 53.455,Y 73.864,Z 70.247,A 180.000,B 0.000,C 180.000} C_DIS
LIN {X 81.433,Y 64.426,Z 70.247,A 180.000,B 0.000,C 180.000} C_DIS
LIN {X 81.478,Y 64.410,Z 70.247,A 180.000,B 0.000,C 180.000} C_DIS
LIN {X 81.500,Y 64.403,Z 70.247,A 180.000,B 0.000,C 180.000} C_DIS
LIN {X 81.522,Y 64.395,Z 70.247,A 180.000,B 0.000,C 180.000} C_DIS
LIN {X 81.545,Y 64.387,Z 70.247,A 180.000,B 0.000,C 180.000} C_DIS
LIN {X 81.567,Y 64.378,Z 70.247,A 180.000,B 0.000,C 180.000} C_DIS
LIN {X 81.590,Y 64.369,Z 70.247,A 180.000,B 0.000,C 180.000} C_DIS
LIN {X 81.612,Y 64.360,Z 70.247,A 180.000,B 0.000,C 180.000} C_DIS
LIN {X 81.634,Y 64.351,Z 70.247,A 180.000,B 0.000,C 180.000} C_DIS
LIN {X 81.657,Y 64.342,Z 70.247,A 180.000,B 0.000,C 180.000} C_DIS
LIN {X 81.701,Y 64.322,Z 70.247,A 180.000,B 0.000,C 180.000} C_DIS
LIN {X 81.746,Y 64.301,Z 70.247,A 180.000,B 0.000,C 180.000} C_DIS
LIN {X 81.790,Y 64.280,Z 70.247,A 180.000,B 0.000,C 180.000} C_DIS
LIN {X 81.835,Y 64.257,Z 70.247,A 180.000,B 0.000,C 180.000} C_DIS
LIN {X 81.880,Y 64.233,Z 70.247,A 180.000,B 0.000,C 180.000} C_DIS
LIN {X 81.924,Y 64.208,Z 70.247,A 180.000,B 0.000,C 180.000} C_DIS
LIN {X 81.968,Y 64.182,Z 70.247,A 180.000,B 0.000,C 180.000} C_DIS
LIN {X 82.013,Y 64.153,Z 70.247,A 180.000,B 0.000,C 180.000} C_DIS
LIN {X 82.059,Y 64.124,Z 70.247,A 180.000,B 0.000,C 180.000} C_DIS
LIN {X 82.142,Y 64.066,Z 70.247,A 180.000,B 0.000,C 180.000} C_DIS
LIN {X 82.225,Y 64.003,Z 70.247,A 180.000,B 0.000,C 180.000} C_DIS
LIN {X 82.237,Y 63.993,Z 70.247,A 180.000,B 0.000,C 180.000} C_DIS
LIN {X 82.327,Y 63.918,Z 70.247,A 180.000,B 0.000,C 180.000} C_DIS
LIN {X 82.416,Y 63.835,Z 70.247,A 180.000,B 0.000,C 180.000} C_DIS
LIN {X 82.427,Y 63.824,Z 70.247,A 180.000,B 0.000,C 180.000} C_DIS
LIN {X 82.591,Y 63.645,Z 70.247,A 180.000,B 0.000,C 180.000} C_DIS
LIN {X 82.595,Y 63.641,Z 70.247,A 180.000,B 0.000,C 180.000} C_DIS
LIN {X 82.727,Y 63.467,Z 70.247,A 180.000,B 0.000,C 180.000} C_DIS
LIN {X 82.774,Y 63.397,Z 70.247,A 180.000,B 0.000,C 180.000} C_DIS
LIN {X 82.840,Y 63.288,Z 70.247,A 180.000,B 0.000,C 180.000} C_DIS
LIN {X 82.933,Y 63.109,Z 70.247,A 180.000,B 0.000,C 180.000} C_DIS
LIN {X 82.940,Y 63.096,Z 70.247,A 180.000,B 0.000,C 180.000} C_DIS
LIN {X 82.946,Y 63.082,Z 70.247,A 180.000,B 0.000,C 180.000} C_DIS
LIN {X 82.948,Y 63.081,Z 70.247,A 180.000,B 0.000,C 180.000} C_DIS
LIN {X 82.952,Y 63.083,Z 70.247,A 180.000,B 0.000,C 180.000} C_DIS
LIN {X 83.002,Y 63.109,Z 70.247,A 180.000,B 0.000,C 180.000} C_DIS
LIN {X 83.131,Y 63.170,Z 70.247,A 180.000,B 0.000,C 180.000} C_DIS
LIN {X 83.310,Y 63.239,Z 70.247,A 180.000,B 0.000,C 180.000} C_DIS
LIN {X 83.466,Y 63.288,Z 70.247,A 180.000,B 0.000,C 180.000} C_DIS
LIN {X 83.489,Y 63.294,Z 70.247,A 180.000,B 0.000,C 180.000} C_DIS
LIN {X 83.668,Y 63.334,Z 70.247,A 180.000,B 0.000,C 180.000} C_DIS
LIN {X 83.846,Y 63.361,Z 70.247,A 180.000,B 0.000,C 180.000} C_DIS
LIN {X 84.025,Y 63.375,Z 70.247,A 180.000,B 0.000,C 180.000} C_DIS
LIN {X 84.114,Y 63.377,Z 70.247,A 180.000,B 0.000,C 180.000} C_DIS
LIN {X 84.204,Y 63.376,Z 70.247,A 180.000,B 0.000,C 180.000} C_DIS
LIN {X 84.293,Y 63.372,Z 70.247,A 180.000,B 0.000,C 180.000} C_DIS
LIN {X 84.383,Y 63.365,Z 70.247,A 180.000,B 0.000,C 180.000} C_DIS
LIN {X 84.427,Y 63.360,Z 70.247,A 180.000,B 0.000,C 180.000} C_DIS
LIN {X 84.472,Y 63.354,Z 70.247,A 180.000,B 0.000,C 180.000} C_DIS
LIN {X 84.517,Y 63.347,Z 70.247,A 180.000,B 0.000,C 180.000} C_DIS
LIN {X 84.561,Y 63.340,Z 70.247,A 180.000,B 0.000,C 180.000} C_DIS
LIN {X 84.606,Y 63.332,Z 70.247,A 180.000,B 0.000,C 180.000} C_DIS
LIN {X 84.651,Y 63.323,Z 70.247,A 180.000,B 0.000,C 180.000} C_DIS
LIN {X 84.695,Y 63.313,Z 70.247,A 180.000,B 0.000,C 180.000} C_DIS
LIN {X 84.740,Y 63.302,Z 70.247,A 180.000,B 0.000,C 180.000} C_DIS
LIN {X 84.767,Y 63.295,Z 70.247,A 180.000,B 0.000,C 180.000} C_DIS
LIN {X 84.793,Y 63.288,Z 70.247,A 180.000,B 0.000,C 180.000} C_DIS
LIN {X 84.825,Y 63.279,Z 70.247,A 180.000,B 0.000,C 180.000} C_DIS
LIN {X 84.856,Y 63.270,Z 70.247,A 180.000,B 0.000,C 180.000} C_DIS
LIN {X 84.887,Y 63.260,Z 70.247,A 180.000,B 0.000,C 180.000} C_DIS
LIN {X 84.919,Y 63.250,Z 70.247,A 180.000,B 0.000,C 180.000} C_DIS
LIN {X 85.098,Y 63.189,Z 70.247,A 180.000,B 0.000,C 180.000} C_DIS
LIN {X 96.464,Y 59.355,Z 70.247,A 180.000,B 0.000,C 180.000} C_DIS
LIN {X 96.539,Y 59.329,Z 70.247,A 180.000,B 0.000,C 180.000} C_DIS
LIN {X 96.718,Y 59.257,Z 70.247,A 180.000,B 0.000,C 180.000} C_DIS
LIN {X 96.883,Y 59.176,Z 70.247,A 180.000,B 0.000,C 180.000} C_DIS
LIN {X 96.897,Y 59.169,Z 70.247,A 180.000,B 0.000,C 180.000} C_DIS
LIN {X 97.075,Y 59.061,Z 70.247,A 180.000,B 0.000,C 180.000} C_DIS
LIN {X 97.167,Y 58.997,Z 70.247,A 180.000,B 0.000,C 180.000} C_DIS
LIN {X 97.254,Y 58.931,Z 70.247,A 180.000,B 0.000,C 180.000} C_DIS
LIN {X 97.385,Y 58.819,Z 70.247,A 180.000,B 0.000,C 180.000} C_DIS
LIN {X 97.433,Y 58.774,Z 70.247,A 180.000,B 0.000,C 180.000} C_DIS
LIN {X 97.562,Y 58.640,Z 70.247,A 180.000,B 0.000,C 180.000} C_DIS
LIN {X 97.612,Y 58.582,Z 70.247,A 180.000,B 0.000,C 180.000} C_DIS
LIN {X 97.707,Y 58.461,Z 70.247,A 180.000,B 0.000,C 180.000} C_DIS
LIN {X 97.790,Y 58.341,Z 70.247,A 180.000,B 0.000,C 180.000} C_DIS
LIN {X 97.828,Y 58.282,Z 70.247,A 180.000,B 0.000,C 180.000} C_DIS
LIN {X 97.928,Y 58.103,Z 70.247,A 180.000,B 0.000,C 180.000} C_DIS
LIN {X 97.969,Y 58.017,Z 70.247,A 180.000,B 0.000,C 180.000} C_DIS
LIN {X 98.009,Y 57.925,Z 70.247,A 180.000,B 0.000,C 180.000} C_DIS
LIN {X 98.075,Y 57.746,Z 70.247,A 180.000,B 0.000,C 180.000} C_DIS
LIN {X 98.125,Y 57.567,Z 70.247,A 180.000,B 0.000,C 180.000} C_DIS
LIN {X 98.148,Y 57.466,Z 70.247,A 180.000,B 0.000,C 180.000} C_DIS
LIN {X 98.162,Y 57.388,Z 70.247,A 180.000,B 0.000,C 180.000} C_DIS
LIN {X 98.186,Y 57.210,Z 70.247,A 180.000,B 0.000,C 180.000} C_DIS
LIN {X 98.196,Y 57.031,Z 70.247,A 180.000,B 0.000,C 180.000} C_DIS
LIN {X 98.193,Y 56.852,Z 70.247,A 180.000,B 0.000,C 180.000} C_DIS
LIN {X 98.178,Y 56.673,Z 70.247,A 180.000,B 0.000,C 180.000} C_DIS
LIN {X 98.150,Y 56.495,Z 70.247,A 180.000,B 0.000,C 180.000} C_DIS
LIN {X 98.148,Y 56.485,Z 70.247,A 180.000,B 0.000,C 180.000} C_DIS
LIN {X 98.108,Y 56.316,Z 70.247,A 180.000,B 0.000,C 180.000} C_DIS
LIN {X 98.052,Y 56.137,Z 70.247,A 180.000,B 0.000,C 180.000} C_DIS
LIN {X 91.712,Y 37.344,Z 70.247,A 180.000,B 0.000,C 180.000} C_DIS
LIN {X 91.659,Y 37.187,Z 70.247,A 180.000,B 0.000,C 180.000} C_DIS
LIN {X 91.588,Y 37.009,Z 70.247,A 180.000,B 0.000,C 180.000} C_DIS
LIN {X 91.533,Y 36.894,Z 70.247,A 180.000,B 0.000,C 180.000} C_DIS
LIN {X 91.500,Y 36.830,Z 70.247,A 180.000,B 0.000,C 180.000} C_DIS
LIN {X 91.392,Y 36.651,Z 70.247,A 180.000,B 0.000,C 180.000} C_DIS
LIN {X 91.355,Y 36.595,Z 70.247,A 180.000,B 0.000,C 180.000} C_DIS
LIN {X 91.263,Y 36.472,Z 70.247,A 180.000,B 0.000,C 180.000} C_DIS
LIN {X 91.176,Y 36.368,Z 70.247,A 180.000,B 0.000,C 180.000} C_DIS
LIN {X 91.107,Y 36.294,Z 70.247,A 180.000,B 0.000,C 180.000} C_DIS
LIN {X 90.997,Y 36.186,Z 70.247,A 180.000,B 0.000,C 180.000} C_DIS
LIN {X 90.917,Y 36.115,Z 70.247,A 180.000,B 0.000,C 180.000} C_DIS
LIN {X 90.818,Y 36.036,Z 70.247,A 180.000,B 0.000,C 180.000} C_DIS
LIN {X 90.677,Y 35.936,Z 70.247,A 180.000,B 0.000,C 180.000} C_DIS
LIN {X 90.640,Y 35.912,Z 70.247,A 180.000,B 0.000,C 180.000} C_DIS
LIN {X 90.461,Y 35.809,Z 70.247,A 180.000,B 0.000,C 180.000} C_DIS
LIN {X 90.356,Y 35.757,Z 70.247,A 180.000,B 0.000,C 180.000} C_DIS
LIN {X 90.282,Y 35.724,Z 70.247,A 180.000,B 0.000,C 180.000} C_DIS
LIN {X 90.103,Y 35.656,Z 70.247,A 180.000,B 0.000,C 180.000} C_DIS
LIN {X 89.925,Y 35.603,Z 70.247,A 180.000,B 0.000,C 180.000} C_DIS
LIN {X 89.819,Y 35.578,Z 70.247,A 180.000,B 0.000,C 180.000} C_DIS
LIN {X 89.746,Y 35.564,Z 70.247,A 180.000,B 0.000,C 180.000} C_DIS
LIN {X 89.567,Y 35.539,Z 70.247,A 180.000,B 0.000,C 180.000} C_DIS
LIN {X 89.388,Y 35.526,Z 70.247,A 180.000,B 0.000,C 180.000} C_DIS
LIN {X 89.209,Y 35.526,Z 70.247,A 180.000,B 0.000,C 180.000} C_DIS
LIN {X 89.031,Y 35.540,Z 70.247,A 180.000,B 0.000,C 180.000} C_DIS
LIN {X 88.852,Y 35.566,Z 70.247,A 180.000,B 0.000,C 180.000} C_DIS
LIN {X 88.788,Y 35.578,Z 70.247,A 180.000,B 0.000,C 180.000} C_DIS
LIN {X 88.673,Y 35.605,Z 70.247,A 180.000,B 0.000,C 180.000} C_DIS
LIN {X 88.494,Y 35.659,Z 70.247,A 180.000,B 0.000,C 180.000} C_DIS
LIN {X 76.964,Y 39.549,Z 70.247,A 180.000,B 0.000,C 180.000} C_DIS
LIN {X 76.919,Y 39.564,Z 70.247,A 180.000,B 0.000,C 180.000} C_DIS
LIN {X 76.897,Y 39.572,Z 70.247,A 180.000,B 0.000,C 180.000} C_DIS
LIN {X 76.874,Y 39.580,Z 70.247,A 180.000,B 0.000,C 180.000} C_DIS
LIN {X 76.852,Y 39.588,Z 70.247,A 180.000,B 0.000,C 180.000} C_DIS
LIN {X 76.830,Y 39.597,Z 70.247,A 180.000,B 0.000,C 180.000} C_DIS
LIN {X 76.807,Y 39.606,Z 70.247,A 180.000,B 0.000,C 180.000} C_DIS
LIN {X 76.785,Y 39.615,Z 70.247,A 180.000,B 0.000,C 180.000} C_DIS
LIN {X 76.740,Y 39.634,Z 70.247,A 180.000,B 0.000,C 180.000} C_DIS
LIN {X 76.696,Y 39.654,Z 70.247,A 180.000,B 0.000,C 180.000} C_DIS
LIN {X 76.658,Y 39.672,Z 70.247,A 180.000,B 0.000,C 180.000} C_DIS
LIN {X 76.620,Y 39.690,Z 70.247,A 180.000,B 0.000,C 180.000} C_DIS
LIN {X 76.568,Y 39.717,Z 70.247,A 180.000,B 0.000,C 180.000} C_DIS
LIN {X 76.517,Y 39.744,Z 70.247,A 180.000,B 0.000,C 180.000} C_DIS
LIN {X 76.472,Y 39.770,Z 70.247,A 180.000,B 0.000,C 180.000} C_DIS
LIN {X 76.427,Y 39.797,Z 70.247,A 180.000,B 0.000,C 180.000} C_DIS
LIN {X 76.338,Y 39.854,Z 70.247,A 180.000,B 0.000,C 180.000} C_DIS
LIN {X 76.317,Y 39.869,Z 70.247,A 180.000,B 0.000,C 180.000} C_DIS
LIN {X 76.238,Y 39.926,Z 70.247,A 180.000,B 0.000,C 180.000} C_DIS
LIN {X 76.159,Y 39.987,Z 70.247,A 180.000,B 0.000,C 180.000} C_DIS
LIN {X 76.087,Y 40.048,Z 70.247,A 180.000,B 0.000,C 180.000} C_DIS
LIN {X 75.980,Y 40.147,Z 70.247,A 180.000,B 0.000,C 180.000} C_DIS
LIN {X 75.904,Y 40.226,Z 70.247,A 180.000,B 0.000,C 180.000} C_DIS
LIN {X 75.802,Y 40.343,Z 70.247,A 180.000,B 0.000,C 180.000} C_DIS
LIN {X 75.753,Y 40.405,Z 70.247,A 180.000,B 0.000,C 180.000} C_DIS
LIN {X 75.628,Y 40.584,Z 70.247,A 180.000,B 0.000,C 180.000} C_DIS
LIN {X 75.623,Y 40.591,Z 70.247,A 180.000,B 0.000,C 180.000} C_DIS
LIN {X 75.524,Y 40.763,Z 70.247,A 180.000,B 0.000,C 180.000} C_DIS
LIN {X 75.494,Y 40.822,Z 70.247,A 180.000,B 0.000,C 180.000} C_DIS
LIN {X 75.479,Y 40.852,Z 70.247,A 180.000,B 0.000,C 180.000} C_DIS
LIN {X 75.462,Y 40.890,Z 70.247,A 180.000,B 0.000,C 180.000} C_DIS
LIN {X 75.460,Y 40.890,Z 70.247,A 180.000,B 0.000,C 180.000} C_DIS
LIN {X 75.453,Y 40.886,Z 70.247,A 180.000,B 0.000,C 180.000} C_DIS
LIN {X 75.444,Y 40.882,Z 70.247,A 180.000,B 0.000,C 180.000} C_DIS
LIN {X 75.265,Y 40.796,Z 70.247,A 180.000,B 0.000,C 180.000} C_DIS
LIN {X 75.184,Y 40.763,Z 70.247,A 180.000,B 0.000,C 180.000} C_DIS
; Link Move Starts
LIN {X 74.999,Y 40.682,Z 70.246,A 180.000,B 0.000,C 180.000} C_DIS
LIN {X 74.818,Y 40.635,Z 70.245,A 180.000,B 0.000,C 180.000} C_DIS
LIN {X 74.649,Y 40.602,Z 70.244,A 180.000,B 0.000,C 180.000} C_DIS
LIN {X 74.478,Y 40.581,Z 70.242,A 180.000,B 0.000,C 180.000} C_DIS
LIN {X 74.397,Y 40.575,Z 70.241,A 180.000,B 0.000,C 180.000} C_DIS
LIN {X 74.316,Y 40.573,Z 70.239,A 180.000,B 0.000,C 180.000} C_DIS
LIN {X 74.235,Y 40.573,Z 70.238,A 180.000,B 0.000,C 180.000} C_DIS
LIN {X 74.154,Y 40.576,Z 70.237,A 180.000,B 0.000,C 180.000} C_DIS
LIN {X 74.077,Y 40.582,Z 70.235,A 180.000,B 0.000,C 180.000} C_DIS
LIN {X 74.038,Y 40.586,Z 70.234,A 180.000,B 0.000,C 180.000} C_DIS
LIN {X 73.999,Y 40.590,Z 70.233,A 180.000,B 0.000,C 180.000} C_DIS
LIN {X 73.961,Y 40.596,Z 70.233,A 180.000,B 0.000,C 180.000} C_DIS
LIN {X 73.922,Y 40.602,Z 70.232,A 180.000,B 0.000,C 180.000} C_DIS
LIN {X 73.884,Y 40.609,Z 70.231,A 180.000,B 0.000,C 180.000} C_DIS
LIN {X 73.846,Y 40.616,Z 70.230,A 180.000,B 0.000,C 180.000} C_DIS
LIN {X 73.808,Y 40.624,Z 70.229,A 180.000,B 0.000,C 180.000} C_DIS
LIN {X 73.771,Y 40.633,Z 70.228,A 180.000,B 0.000,C 180.000} C_DIS
LIN {X 73.734,Y 40.643,Z 70.227,A 180.000,B 0.000,C 180.000} C_DIS
LIN {X 73.698,Y 40.653,Z 70.226,A 180.000,B 0.000,C 180.000} C_DIS
LIN {X 73.679,Y 40.658,Z 70.226,A 180.000,B 0.000,C 180.000} C_DIS
LIN {X 73.661,Y 40.664,Z 70.225,A 180.000,B 0.000,C 180.000} C_DIS
LIN {X 73.643,Y 40.670,Z 70.225,A 180.000,B 0.000,C 180.000} C_DIS
LIN {X 73.625,Y 40.676,Z 70.224,A 180.000,B 0.000,C 180.000} C_DIS
LIN {X 73.552,Y 40.700,Z 70.222,A 180.000,B 0.000,C 180.000} C_DIS
LIN {X 73.408,Y 40.749,Z 70.218,A 180.000,B 0.000,C 180.000} C_DIS
LIN {X 73.263,Y 40.798,Z 70.214,A 180.000,B 0.000,C 180.000} C_DIS
LIN {X 73.118,Y 40.846,Z 70.209,A 180.000,B 0.000,C 180.000} C_DIS
LIN {X 73.046,Y 40.871,Z 70.206,A 180.000,B 0.000,C 180.000} C_DIS
LIN {X 72.974,Y 40.895,Z 70.204,A 180.000,B 0.000,C 180.000} C_DIS
LIN {X 72.901,Y 40.919,Z 70.201,A 180.000,B 0.000,C 180.000} C_DIS
LIN {X 72.829,Y 40.944,Z 70.198,A 180.000,B 0.000,C 180.000} C_DIS
LIN {X 72.757,Y 40.968,Z 70.196,A 180.000,B 0.000,C 180.000} C_DIS
LIN {X 72.685,Y 40.993,Z 70.193,A 180.000,B 0.000,C 180.000} C_DIS
LIN {X 72.612,Y 41.017,Z 70.190,A 180.000,B 0.000,C 180.000} C_DIS
LIN {X 72.540,Y 41.041,Z 70.188,A 180.000,B 0.000,C 180.000} C_DIS
LIN {X 72.468,Y 41.066,Z 70.185,A 180.000,B 0.000,C 180.000} C_DIS
LIN {X 72.395,Y 41.090,Z 70.182,A 180.000,B 0.000,C 180.000} C_DIS
LIN {X 72.323,Y 41.115,Z 70.180,A 180.000,B 0.000,C 180.000} C_DIS
LIN {X 72.251,Y 41.139,Z 70.177,A 180.000,B 0.000,C 180.000} C_DIS
LIN {X 72.179,Y 41.163,Z 70.174,A 180.000,B 0.000,C 180.000} C_DIS
LIN {X 72.106,Y 41.188,Z 70.172,A 180.000,B 0.000,C 180.000} C_DIS
LIN {X 72.034,Y 41.212,Z 70.169,A 180.000,B 0.000,C 180.000} C_DIS
LIN {X 71.962,Y 41.236,Z 70.166,A 180.000,B 0.000,C 180.000} C_DIS
LIN {X 71.889,Y 41.261,Z 70.164,A 180.000,B 0.000,C 180.000} C_DIS
LIN {X 71.817,Y 41.285,Z 70.161,A 180.000,B 0.000,C 180.000} C_DIS
LIN {X 71.745,Y 41.310,Z 70.158,A 180.000,B 0.000,C 180.000} C_DIS
LIN {X 71.600,Y 41.358,Z 70.153,A 180.000,B 0.000,C 180.000} C_DIS
LIN {X 71.528,Y 41.383,Z 70.150,A 180.000,B 0.000,C 180.000} C_DIS
LIN {X 71.383,Y 41.432,Z 70.145,A 180.000,B 0.000,C 180.000} C_DIS
LIN {X 71.094,Y 41.529,Z 70.134,A 180.000,B 0.000,C 180.000} C_DIS
LIN {X 70.444,Y 41.749,Z 70.110,A 180.000,B 0.000,C 180.000} C_DIS
LIN {X 70.371,Y 41.773,Z 70.108,A 180.000,B 0.000,C 180.000} C_DIS
LIN {X 70.227,Y 41.822,Z 70.102,A 180.000,B 0.000,C 180.000} C_DIS
LIN {X 70.010,Y 41.895,Z 70.094,A 180.000,B 0.000,C 180.000} C_DIS
LIN {X 69.865,Y 41.944,Z 70.089,A 180.000,B 0.000,C 180.000} C_DIS
LIN {X 69.793,Y 41.968,Z 70.086,A 180.000,B 0.000,C 180.000} C_DIS
LIN {X 69.721,Y 41.992,Z 70.084,A 180.000,B 0.000,C 180.000} C_DIS
LIN {X 69.648,Y 42.017,Z 70.081,A 180.000,B 0.000,C 180.000} C_DIS
LIN {X 69.576,Y 42.041,Z 70.078,A 180.000,B 0.000,C 180.000} C_DIS
LIN {X 69.504,Y 42.066,Z 70.076,A 180.000,B 0.000,C 180.000} C_DIS
LIN {X 69.432,Y 42.090,Z 70.073,A 180.000,B 0.000,C 180.000} C_DIS
LIN {X 69.359,Y 42.114,Z 70.070,A 180.000,B 0.000,C 180.000} C_DIS
LIN {X 69.287,Y 42.139,Z 70.068,A 180.000,B 0.000,C 180.000} C_DIS
LIN {X 69.215,Y 42.163,Z 70.065,A 180.000,B 0.000,C 180.000} C_DIS
LIN {X 69.142,Y 42.188,Z 70.062,A 180.000,B 0.000,C 180.000} C_DIS
LIN {X 69.070,Y 42.212,Z 70.060,A 180.000,B 0.000,C 180.000} C_DIS
LIN {X 68.998,Y 42.236,Z 70.057,A 180.000,B 0.000,C 180.000} C_DIS
LIN {X 68.926,Y 42.261,Z 70.055,A 180.000,B 0.000,C 180.000} C_DIS
LIN {X 68.853,Y 42.285,Z 70.052,A 180.000,B 0.000,C 180.000} C_DIS
LIN {X 68.781,Y 42.309,Z 70.049,A 180.000,B 0.000,C 180.000} C_DIS
LIN {X 68.709,Y 42.334,Z 70.046,A 180.000,B 0.000,C 180.000} C_DIS
LIN {X 68.636,Y 42.358,Z 70.044,A 180.000,B 0.000,C 180.000} C_DIS
LIN {X 68.564,Y 42.383,Z 70.041,A 180.000,B 0.000,C 180.000} C_DIS
LIN {X 68.492,Y 42.407,Z 70.039,A 180.000,B 0.000,C 180.000} C_DIS
LIN {X 68.347,Y 42.456,Z 70.034,A 180.000,B 0.000,C 180.000} C_DIS
LIN {X 68.203,Y 42.505,Z 70.029,A 180.000,B 0.000,C 180.000} C_DIS
LIN {X 68.058,Y 42.553,Z 70.025,A 180.000,B 0.000,C 180.000} C_DIS
LIN {X 67.914,Y 42.602,Z 70.021,A 180.000,B 0.000,C 180.000} C_DIS
LIN {X 67.769,Y 42.651,Z 70.017,A 180.000,B 0.000,C 180.000} C_DIS
LIN {X 67.624,Y 42.700,Z 70.014,A 180.000,B 0.000,C 180.000} C_DIS
LIN {X 67.480,Y 42.748,Z 70.011,A 180.000,B 0.000,C 180.000} C_DIS
LIN {X 67.335,Y 42.797,Z 70.008,A 180.000,B 0.000,C 180.000} C_DIS
LIN {X 67.191,Y 42.846,Z 70.006,A 180.000,B 0.000,C 180.000} C_DIS
LIN {X 66.901,Y 42.944,Z 70.002,A 180.000,B 0.000,C 180.000} C_DIS
LIN {X 66.612,Y 43.041,Z 70.000,A 180.000,B 0.000,C 180.000} C_DIS
LIN {X 66.460,Y 43.092,Z 70.000,A 180.000,B 0.000,C 180.000} C_DIS
; Cutting Move Starts
LIN {X 45.590,Y 50.133,Z 70.000,A 180.000,B 0.000,C 180.000} C_DIS
LIN {X 45.411,Y 50.194,Z 70.000,A 180.000,B 0.000,C 180.000} C_DIS
LIN {X 45.296,Y 50.238,Z 70.000,A 180.000,B 0.000,C 180.000} C_DIS
LIN {X 45.232,Y 50.265,Z 70.000,A 180.000,B 0.000,C 180.000} C_DIS
LIN {X 45.053,Y 50.353,Z 70.000,A 180.000,B 0.000,C 180.000} C_DIS
LIN {X 44.944,Y 50.416,Z 70.000,A 180.000,B 0.000,C 180.000} C_DIS
LIN {X 44.874,Y 50.461,Z 70.000,A 180.000,B 0.000,C 180.000} C_DIS
LIN {X 44.785,Y 50.522,Z 70.000,A 180.000,B 0.000,C 180.000} C_DIS
LIN {X 44.696,Y 50.590,Z 70.000,A 180.000,B 0.000,C 180.000} C_DIS
LIN {X 44.689,Y 50.595,Z 70.000,A 180.000,B 0.000,C 180.000} C_DIS
LIN {X 44.603,Y 50.667,Z 70.000,A 180.000,B 0.000,C 180.000} C_DIS
LIN {X 44.517,Y 50.746,Z 70.000,A 180.000,B 0.000,C 180.000} C_DIS
LIN {X 44.488,Y 50.774,Z 70.000,A 180.000,B 0.000,C 180.000} C_DIS
LIN {X 44.410,Y 50.855,Z 70.000,A 180.000,B 0.000,C 180.000} C_DIS
LIN {X 44.338,Y 50.936,Z 70.000,A 180.000,B 0.000,C 180.000} C_DIS
LIN {X 44.325,Y 50.953,Z 70.000,A 180.000,B 0.000,C 180.000} C_DIS
LIN {X 44.254,Y 51.042,Z 70.000,A 180.000,B 0.000,C 180.000} C_DIS
LIN {X 44.189,Y 51.131,Z 70.000,A 180.000,B 0.000,C 180.000} C_DIS
LIN {X 44.159,Y 51.176,Z 70.000,A 180.000,B 0.000,C 180.000} C_DIS
LIN {X 44.077,Y 51.310,Z 70.000,A 180.000,B 0.000,C 180.000} C_DIS
LIN {X 43.984,Y 51.489,Z 70.000,A 180.000,B 0.000,C 180.000} C_DIS
LIN {X 43.981,Y 51.497,Z 70.000,A 180.000,B 0.000,C 180.000} C_DIS
LIN {X 43.909,Y 51.668,Z 70.000,A 180.000,B 0.000,C 180.000} C_DIS
LIN {X 43.849,Y 51.847,Z 70.000,A 180.000,B 0.000,C 180.000} C_DIS
LIN {X 43.804,Y 52.025,Z 70.000,A 180.000,B 0.000,C 180.000} C_DIS
LIN {X 43.802,Y 52.035,Z 70.000,A 180.000,B 0.000,C 180.000} C_DIS
LIN {X 43.772,Y 52.204,Z 70.000,A 180.000,B 0.000,C 180.000} C_DIS
LIN {X 43.754,Y 52.383,Z 70.000,A 180.000,B 0.000,C 180.000} C_DIS
LIN {X 43.748,Y 52.562,Z 70.000,A 180.000,B 0.000,C 180.000} C_DIS
LIN {X 43.756,Y 52.740,Z 70.000,A 180.000,B 0.000,C 180.000} C_DIS
LIN {X 43.776,Y 52.919,Z 70.000,A 180.000,B 0.000,C 180.000} C_DIS
LIN {X 43.802,Y 53.064,Z 70.000,A 180.000,B 0.000,C 180.000} C_DIS
LIN {X 43.809,Y 53.098,Z 70.000,A 180.000,B 0.000,C 180.000} C_DIS
LIN {X 43.856,Y 53.277,Z 70.000,A 180.000,B 0.000,C 180.000} C_DIS
LIN {X 43.916,Y 53.455,Z 70.000,A 180.000,B 0.000,C 180.000} C_DIS
LIN {X 50.248,Y 72.226,Z 70.000,A 180.000,B 0.000,C 180.000} C_DIS
LIN {X 50.311,Y 72.405,Z 70.000,A 180.000,B 0.000,C 180.000} C_DIS
LIN {X 50.388,Y 72.584,Z 70.000,A 180.000,B 0.000,C 180.000} C_DIS
LIN {X 50.416,Y 72.640,Z 70.000,A 180.000,B 0.000,C 180.000} C_DIS
LIN {X 50.484,Y 72.763,Z 70.000,A 180.000,B 0.000,C 180.000} C_DIS
LIN {X 50.595,Y 72.936,Z 70.000,A 180.000,B 0.000,C 180.000} C_DIS
LIN {X 50.599,Y 72.941,Z 70.000,A 180.000,B 0.000,C 180.000} C_DIS
LIN {X 50.665,Y 73.031,Z 70.000,A 180.000,B 0.000,C 180.000} C_DIS
LIN {X 50.737,Y 73.120,Z 70.000,A 180.000,B 0.000,C 180.000} C_DIS
LIN {X 50.774,Y 73.162,Z 70.000,A 180.000,B 0.000,C 180.000} C_DIS
LIN {X 50.905,Y 73.299,Z 70.000,A 180.000,B 0.000,C 180.000} C_DIS
LIN {X 50.953,Y 73.343,Z 70.000,A 180.000,B 0.000,C 180.000} C_DIS
LIN {X 51.112,Y 73.478,Z 70.000,A 180.000,B 0.000,C 180.000} C_DIS
LIN {X 51.131,Y 73.493,Z 70.000,A 180.000,B 0.000,C 180.000} C_DIS
LIN {X 51.310,Y 73.616,Z 70.000,A 180.000,B 0.000,C 180.000} C_DIS
LIN {X 51.376,Y 73.656,Z 70.000,A 180.000,B 0.000,C 180.000} C_DIS
LIN {X 51.489,Y 73.719,Z 70.000,A 180.000,B 0.000,C 180.000} C_DIS
LIN {X 51.668,Y 73.803,Z 70.000,A 180.000,B 0.000,C 180.000} C_DIS
LIN {X 51.749,Y 73.835,Z 70.000,A 180.000,B 0.000,C 180.000} C_DIS
LIN {X 51.847,Y 73.870,Z 70.000,A 180.000,B 0.000,C 180.000} C_DIS
LIN {X 52.025,Y 73.923,Z 70.000,A 180.000,B 0.000,C 180.000} C_DIS
LIN {X 52.204,Y 73.961,Z 70.000,A 180.000,B 0.000,C 180.000} C_DIS
LIN {X 52.383,Y 73.987,Z 70.000,A 180.000,B 0.000,C 180.000} C_DIS
LIN {X 52.562,Y 73.999,Z 70.000,A 180.000,B 0.000,C 180.000} C_DIS
LIN {X 52.740,Y 73.998,Z 70.000,A 180.000,B 0.000,C 180.000} C_DIS
LIN {X 52.919,Y 73.985,Z 70.000,A 180.000,B 0.000,C 180.000} C_DIS
LIN {X 53.098,Y 73.958,Z 70.000,A 180.000,B 0.000,C 180.000} C_DIS
LIN {X 53.277,Y 73.918,Z 70.000,A 180.000,B 0.000,C 180.000} C_DIS
LIN {X 53.455,Y 73.864,Z 70.000,A 180.000,B 0.000,C 180.000} C_DIS
LIN {X 83.198,Y 63.830,Z 70.000,A 180.000,B 0.000,C 180.000} C_DIS
LIN {X 96.464,Y 59.355,Z 70.000,A 180.000,B 0.000,C 180.000} C_DIS
LIN {X 96.539,Y 59.329,Z 70.000,A 180.000,B 0.000,C 180.000} C_DIS
LIN {X 96.718,Y 59.257,Z 70.000,A 180.000,B 0.000,C 180.000} C_DIS
LIN {X 96.883,Y 59.176,Z 70.000,A 180.000,B 0.000,C 180.000} C_DIS
LIN {X 96.897,Y 59.169,Z 70.000,A 180.000,B 0.000,C 180.000} C_DIS
LIN {X 97.075,Y 59.061,Z 70.000,A 180.000,B 0.000,C 180.000} C_DIS
LIN {X 97.167,Y 58.997,Z 70.000,A 180.000,B 0.000,C 180.000} C_DIS
LIN {X 97.254,Y 58.931,Z 70.000,A 180.000,B 0.000,C 180.000} C_DIS
LIN {X 97.385,Y 58.819,Z 70.000,A 180.000,B 0.000,C 180.000} C_DIS
LIN {X 97.433,Y 58.774,Z 70.000,A 180.000,B 0.000,C 180.000} C_DIS
LIN {X 97.562,Y 58.640,Z 70.000,A 180.000,B 0.000,C 180.000} C_DIS
LIN {X 97.612,Y 58.582,Z 70.000,A 180.000,B 0.000,C 180.000} C_DIS
LIN {X 97.707,Y 58.461,Z 70.000,A 180.000,B 0.000,C 180.000} C_DIS
LIN {X 97.790,Y 58.341,Z 70.000,A 180.000,B 0.000,C 180.000} C_DIS
LIN {X 97.828,Y 58.282,Z 70.000,A 180.000,B 0.000,C 180.000} C_DIS
LIN {X 97.928,Y 58.103,Z 70.000,A 180.000,B 0.000,C 180.000} C_DIS
LIN {X 97.969,Y 58.017,Z 70.000,A 180.000,B 0.000,C 180.000} C_DIS
LIN {X 98.009,Y 57.925,Z 70.000,A 180.000,B 0.000,C 180.000} C_DIS
LIN {X 98.075,Y 57.746,Z 70.000,A 180.000,B 0.000,C 180.000} C_DIS
LIN {X 98.125,Y 57.567,Z 70.000,A 180.000,B 0.000,C 180.000} C_DIS
LIN {X 98.148,Y 57.466,Z 70.000,A 180.000,B 0.000,C 180.000} C_DIS
LIN {X 98.162,Y 57.388,Z 70.000,A 180.000,B 0.000,C 180.000} C_DIS
LIN {X 98.186,Y 57.210,Z 70.000,A 180.000,B 0.000,C 180.000} C_DIS
LIN {X 98.196,Y 57.031,Z 70.000,A 180.000,B 0.000,C 180.000} C_DIS
LIN {X 98.193,Y 56.852,Z 70.000,A 180.000,B 0.000,C 180.000} C_DIS
LIN {X 98.178,Y 56.673,Z 70.000,A 180.000,B 0.000,C 180.000} C_DIS
LIN {X 98.150,Y 56.495,Z 70.000,A 180.000,B 0.000,C 180.000} C_DIS
LIN {X 98.148,Y 56.485,Z 70.000,A 180.000,B 0.000,C 180.000} C_DIS
LIN {X 98.108,Y 56.316,Z 70.000,A 180.000,B 0.000,C 180.000} C_DIS
LIN {X 98.052,Y 56.137,Z 70.000,A 180.000,B 0.000,C 180.000} C_DIS
LIN {X 97.062,Y 53.202,Z 70.000,A 180.000,B 0.000,C 180.000} C_DIS
LIN {X 97.064,Y 53.200,Z 70.000,A 180.000,B 0.000,C 180.000} C_DIS
LIN {X 97.075,Y 53.191,Z 70.000,A 180.000,B 0.000,C 180.000} C_DIS
LIN {X 97.192,Y 53.098,Z 70.000,A 180.000,B 0.000,C 180.000} C_DIS
LIN {X 97.254,Y 53.045,Z 70.000,A 180.000,B 0.000,C 180.000} C_DIS
LIN {X 97.394,Y 52.919,Z 70.000,A 180.000,B 0.000,C 180.000} C_DIS
LIN {X 97.433,Y 52.884,Z 70.000,A 180.000,B 0.000,C 180.000} C_DIS
LIN {X 97.588,Y 52.740,Z 70.000,A 180.000,B 0.000,C 180.000} C_DIS
LIN {X 97.612,Y 52.717,Z 70.000,A 180.000,B 0.000,C 180.000} C_DIS
LIN {X 97.790,Y 52.534,Z 70.000,A 180.000,B 0.000,C 180.000} C_DIS
LIN {X 97.931,Y 52.383,Z 70.000,A 180.000,B 0.000,C 180.000} C_DIS
LIN {X 98.086,Y 52.204,Z 70.000,A 180.000,B 0.000,C 180.000} C_DIS
LIN {X 98.148,Y 52.131,Z 70.000,A 180.000,B 0.000,C 180.000} C_DIS
LIN {X 98.233,Y 52.025,Z 70.000,A 180.000,B 0.000,C 180.000} C_DIS
LIN {X 98.368,Y 51.847,Z 70.000,A 180.000,B 0.000,C 180.000} C_DIS
LIN {X 98.498,Y 51.668,Z 70.000,A 180.000,B 0.000,C 180.000} C_DIS
LIN {X 98.505,Y 51.656,Z 70.000,A 180.000,B 0.000,C 180.000} C_DIS
LIN {X 98.616,Y 51.489,Z 70.000,A 180.000,B 0.000,C 180.000} C_DIS
LIN {X 98.684,Y 51.386,Z 70.000,A 180.000,B 0.000,C 180.000} C_DIS
LIN {X 98.732,Y 51.310,Z 70.000,A 180.000,B 0.000,C 180.000} C_DIS
LIN {X 98.835,Y 51.131,Z 70.000,A 180.000,B 0.000,C 180.000} C_DIS
LIN {X 98.863,Y 51.083,Z 70.000,A 180.000,B 0.000,C 180.000} C_DIS
LIN {X 98.937,Y 50.953,Z 70.000,A 180.000,B 0.000,C 180.000} C_DIS
LIN {X 99.027,Y 50.774,Z 70.000,A 180.000,B 0.000,C 180.000} C_DIS
LIN {X 99.042,Y 50.744,Z 70.000,A 180.000,B 0.000,C 180.000} C_DIS
LIN {X 99.116,Y 50.595,Z 70.000,A 180.000,B 0.000,C 180.000} C_DIS
LIN {X 99.195,Y 50.416,Z 70.000,A 180.000,B 0.000,C 180.000} C_DIS
LIN {X 99.270,Y 50.238,Z 70.000,A 180.000,B 0.000,C 180.000} C_DIS
LIN {X 99.341,Y 50.059,Z 70.000,A 180.000,B 0.000,C 180.000} C_DIS
LIN {X 99.399,Y 49.891,Z 70.000,A 180.000,B 0.000,C 180.000} C_DIS
LIN {X 99.403,Y 49.880,Z 70.000,A 180.000,B 0.000,C 180.000} C_DIS
LIN {X 99.465,Y 49.701,Z 70.000,A 180.000,B 0.000,C 180.000} C_DIS
LIN {X 99.517,Y 49.523,Z 70.000,A 180.000,B 0.000,C 180.000} C_DIS
LIN {X 99.566,Y 49.344,Z 70.000,A 180.000,B 0.000,C 180.000} C_DIS
LIN {X 99.578,Y 49.302,Z 70.000,A 180.000,B 0.000,C 180.000} C_DIS
LIN {X 99.611,Y 49.165,Z 70.000,A 180.000,B 0.000,C 180.000} C_DIS
LIN {X 99.649,Y 48.986,Z 70.000,A 180.000,B 0.000,C 180.000} C_DIS
LIN {X 99.686,Y 48.807,Z 70.000,A 180.000,B 0.000,C 180.000} C_DIS
LIN {X 99.715,Y 48.629,Z 70.000,A 180.000,B 0.000,C 180.000} C_DIS
LIN {X 99.741,Y 48.450,Z 70.000,A 180.000,B 0.000,C 180.000} C_DIS
LIN {X 99.757,Y 48.332,Z 70.000,A 180.000,B 0.000,C 180.000} C_DIS
LIN {X 99.763,Y 48.271,Z 70.000,A 180.000,B 0.000,C 180.000} C_DIS
LIN {X 99.778,Y 48.092,Z 70.000,A 180.000,B 0.000,C 180.000} C_DIS
LIN {X 99.792,Y 47.914,Z 70.000,A 180.000,B 0.000,C 180.000} C_DIS
LIN {X 99.799,Y 47.735,Z 70.000,A 180.000,B 0.000,C 180.000} C_DIS
LIN {X 99.802,Y 47.556,Z 70.000,A 180.000,B 0.000,C 180.000} C_DIS
LIN {X 99.803,Y 47.377,Z 70.000,A 180.000,B 0.000,C 180.000} C_DIS
LIN {X 99.796,Y 47.198,Z 70.000,A 180.000,B 0.000,C 180.000} C_DIS
LIN {X 99.788,Y 47.020,Z 70.000,A 180.000,B 0.000,C 180.000} C_DIS
LIN {X 99.773,Y 46.841,Z 70.000,A 180.000,B 0.000,C 180.000} C_DIS
LIN {X 99.754,Y 46.662,Z 70.000,A 180.000,B 0.000,C 180.000} C_DIS
LIN {X 99.733,Y 46.483,Z 70.000,A 180.000,B 0.000,C 180.000} C_DIS
LIN {X 99.704,Y 46.305,Z 70.000,A 180.000,B 0.000,C 180.000} C_DIS
LIN {X 99.673,Y 46.126,Z 70.000,A 180.000,B 0.000,C 180.000} C_DIS
LIN {X 99.636,Y 45.947,Z 70.000,A 180.000,B 0.000,C 180.000} C_DIS
LIN {X 99.578,Y 45.701,Z 70.000,A 180.000,B 0.000,C 180.000} C_DIS
LIN {X 99.550,Y 45.590,Z 70.000,A 180.000,B 0.000,C 180.000} C_DIS
LIN {X 99.497,Y 45.411,Z 70.000,A 180.000,B 0.000,C 180.000} C_DIS
LIN {X 99.443,Y 45.232,Z 70.000,A 180.000,B 0.000,C 180.000} C_DIS
LIN {X 99.399,Y 45.103,Z 70.000,A 180.000,B 0.000,C 180.000} C_DIS
LIN {X 99.381,Y 45.053,Z 70.000,A 180.000,B 0.000,C 180.000} C_DIS
LIN {X 99.314,Y 44.874,Z 70.000,A 180.000,B 0.000,C 180.000} C_DIS
LIN {X 99.244,Y 44.696,Z 70.000,A 180.000,B 0.000,C 180.000} C_DIS
LIN {X 99.221,Y 44.642,Z 70.000,A 180.000,B 0.000,C 180.000} C_DIS
LIN {X 99.165,Y 44.517,Z 70.000,A 180.000,B 0.000,C 180.000} C_DIS
LIN {X 99.084,Y 44.338,Z 70.000,A 180.000,B 0.000,C 180.000} C_DIS
LIN {X 99.042,Y 44.252,Z 70.000,A 180.000,B 0.000,C 180.000} C_DIS
LIN {X 98.993,Y 44.159,Z 70.000,A 180.000,B 0.000,C 180.000} C_DIS
LIN {X 98.900,Y 43.981,Z 70.000,A 180.000,B 0.000,C 180.000} C_DIS
LIN {X 98.863,Y 43.913,Z 70.000,A 180.000,B 0.000,C 180.000} C_DIS
LIN {X 98.797,Y 43.802,Z 70.000,A 180.000,B 0.000,C 180.000} C_DIS
LIN {X 98.684,Y 43.616,Z 70.000,A 180.000,B 0.000,C 180.000} C_DIS
LIN {X 98.574,Y 43.444,Z 70.000,A 180.000,B 0.000,C 180.000} C_DIS
LIN {X 98.449,Y 43.266,Z 70.000,A 180.000,B 0.000,C 180.000} C_DIS
LIN {X 98.327,Y 43.096,Z 70.000,A 180.000,B 0.000,C 180.000} C_DIS
LIN {X 98.320,Y 43.087,Z 70.000,A 180.000,B 0.000,C 180.000} C_DIS
LIN {X 98.148,Y 42.870,Z 70.000,A 180.000,B 0.000,C 180.000} C_DIS
LIN {X 98.030,Y 42.729,Z 70.000,A 180.000,B 0.000,C 180.000} C_DIS
LIN {X 97.969,Y 42.661,Z 70.000,A 180.000,B 0.000,C 180.000} C_DIS
LIN {X 97.869,Y 42.550,Z 70.000,A 180.000,B 0.000,C 180.000} C_DIS
LIN {X 97.790,Y 42.464,Z 70.000,A 180.000,B 0.000,C 180.000} C_DIS
LIN {X 97.700,Y 42.372,Z 70.000,A 180.000,B 0.000,C 180.000} C_DIS
LIN {X 97.517,Y 42.193,Z 70.000,A 180.000,B 0.000,C 180.000} C_DIS
LIN {X 97.433,Y 42.113,Z 70.000,A 180.000,B 0.000,C 180.000} C_DIS
LIN {X 97.320,Y 42.014,Z 70.000,A 180.000,B 0.000,C 180.000} C_DIS
LIN {X 97.254,Y 41.958,Z 70.000,A 180.000,B 0.000,C 180.000} C_DIS
LIN {X 97.111,Y 41.835,Z 70.000,A 180.000,B 0.000,C 180.000} C_DIS
LIN {X 97.075,Y 41.806,Z 70.000,A 180.000,B 0.000,C 180.000} C_DIS
LIN {X 96.897,Y 41.670,Z 70.000,A 180.000,B 0.000,C 180.000} C_DIS
LIN {X 96.879,Y 41.657,Z 70.000,A 180.000,B 0.000,C 180.000} C_DIS
LIN {X 96.718,Y 41.536,Z 70.000,A 180.000,B 0.000,C 180.000} C_DIS
LIN {X 96.631,Y 41.478,Z 70.000,A 180.000,B 0.000,C 180.000} C_DIS
LIN {X 96.539,Y 41.417,Z 70.000,A 180.000,B 0.000,C 180.000} C_DIS
LIN {X 96.360,Y 41.299,Z 70.000,A 180.000,B 0.000,C 180.000} C_DIS
LIN {X 96.181,Y 41.194,Z 70.000,A 180.000,B 0.000,C 180.000} C_DIS
LIN {X 96.054,Y 41.120,Z 70.000,A 180.000,B 0.000,C 180.000} C_DIS
LIN {X 96.003,Y 41.091,Z 70.000,A 180.000,B 0.000,C 180.000} C_DIS
LIN {X 95.824,Y 40.998,Z 70.000,A 180.000,B 0.000,C 180.000} C_DIS
LIN {X 95.645,Y 40.909,Z 70.000,A 180.000,B 0.000,C 180.000} C_DIS
LIN {X 95.466,Y 40.826,Z 70.000,A 180.000,B 0.000,C 180.000} C_DIS
LIN {X 95.288,Y 40.751,Z 70.000,A 180.000,B 0.000,C 180.000} C_DIS
LIN {X 95.109,Y 40.677,Z 70.000,A 180.000,B 0.000,C 180.000} C_DIS
LIN {X 94.930,Y 40.614,Z 70.000,A 180.000,B 0.000,C 180.000} C_DIS
LIN {X 94.751,Y 40.552,Z 70.000,A 180.000,B 0.000,C 180.000} C_DIS
LIN {X 94.573,Y 40.497,Z 70.000,A 180.000,B 0.000,C 180.000} C_DIS
LIN {X 94.394,Y 40.448,Z 70.000,A 180.000,B 0.000,C 180.000} C_DIS
LIN {X 94.237,Y 40.405,Z 70.000,A 180.000,B 0.000,C 180.000} C_DIS
LIN {X 94.215,Y 40.400,Z 70.000,A 180.000,B 0.000,C 180.000} C_DIS
LIN {X 94.036,Y 40.361,Z 70.000,A 180.000,B 0.000,C 180.000} C_DIS
LIN {X 93.857,Y 40.324,Z 70.000,A 180.000,B 0.000,C 180.000} C_DIS
LIN {X 93.679,Y 40.293,Z 70.000,A 180.000,B 0.000,C 180.000} C_DIS
LIN {X 93.500,Y 40.267,Z 70.000,A 180.000,B 0.000,C 180.000} C_DIS
LIN {X 93.321,Y 40.242,Z 70.000,A 180.000,B 0.000,C 180.000} C_DIS
LIN {X 93.145,Y 40.226,Z 70.000,A 180.000,B 0.000,C 180.000} C_DIS
LIN {X 92.964,Y 40.211,Z 70.000,A 180.000,B 0.000,C 180.000} C_DIS
LIN {X 92.785,Y 40.202,Z 70.000,A 180.000,B 0.000,C 180.000} C_DIS
LIN {X 92.677,Y 40.200,Z 70.000,A 180.000,B 0.000,C 180.000} C_DIS
LIN {X 92.675,Y 40.198,Z 70.000,A 180.000,B 0.000,C 180.000} C_DIS
LIN {X 91.712,Y 37.344,Z 70.000,A 180.000,B 0.000,C 180.000} C_DIS
LIN {X 91.659,Y 37.187,Z 70.000,A 180.000,B 0.000,C 180.000} C_DIS
LIN {X 91.588,Y 37.009,Z 70.000,A 180.000,B 0.000,C 180.000} C_DIS
LIN {X 91.533,Y 36.894,Z 70.000,A 180.000,B 0.000,C 180.000} C_DIS
LIN {X 91.500,Y 36.830,Z 70.000,A 180.000,B 0.000,C 180.000} C_DIS
LIN {X 91.392,Y 36.651,Z 70.000,A 180.000,B 0.000,C 180.000} C_DIS
LIN {X 91.355,Y 36.595,Z 70.000,A 180.000,B 0.000,C 180.000} C_DIS
LIN {X 91.263,Y 36.472,Z 70.000,A 180.000,B 0.000,C 180.000} C_DIS
LIN {X 91.176,Y 36.368,Z 70.000,A 180.000,B 0.000,C 180.000} C_DIS
LIN {X 91.107,Y 36.294,Z 70.000,A 180.000,B 0.000,C 180.000} C_DIS
LIN {X 90.997,Y 36.186,Z 70.000,A 180.000,B 0.000,C 180.000} C_DIS
LIN {X 90.917,Y 36.115,Z 70.000,A 180.000,B 0.000,C 180.000} C_DIS
LIN {X 90.818,Y 36.036,Z 70.000,A 180.000,B 0.000,C 180.000} C_DIS
LIN {X 90.677,Y 35.936,Z 70.000,A 180.000,B 0.000,C 180.000} C_DIS
LIN {X 90.640,Y 35.912,Z 70.000,A 180.000,B 0.000,C 180.000} C_DIS
LIN {X 90.461,Y 35.809,Z 70.000,A 180.000,B 0.000,C 180.000} C_DIS
LIN {X 90.356,Y 35.757,Z 70.000,A 180.000,B 0.000,C 180.000} C_DIS
LIN {X 90.282,Y 35.724,Z 70.000,A 180.000,B 0.000,C 180.000} C_DIS
LIN {X 90.103,Y 35.656,Z 70.000,A 180.000,B 0.000,C 180.000} C_DIS
LIN {X 89.925,Y 35.603,Z 70.000,A 180.000,B 0.000,C 180.000} C_DIS
LIN {X 89.819,Y 35.578,Z 70.000,A 180.000,B 0.000,C 180.000} C_DIS
LIN {X 89.746,Y 35.564,Z 70.000,A 180.000,B 0.000,C 180.000} C_DIS
LIN {X 89.567,Y 35.539,Z 70.000,A 180.000,B 0.000,C 180.000} C_DIS
LIN {X 89.388,Y 35.526,Z 70.000,A 180.000,B 0.000,C 180.000} C_DIS
LIN {X 89.209,Y 35.526,Z 70.000,A 180.000,B 0.000,C 180.000} C_DIS
LIN {X 89.031,Y 35.540,Z 70.000,A 180.000,B 0.000,C 180.000} C_DIS
LIN {X 88.852,Y 35.566,Z 70.000,A 180.000,B 0.000,C 180.000} C_DIS
LIN {X 88.788,Y 35.578,Z 70.000,A 180.000,B 0.000,C 180.000} C_DIS
LIN {X 88.673,Y 35.605,Z 70.000,A 180.000,B 0.000,C 180.000} C_DIS
LIN {X 88.494,Y 35.659,Z 70.000,A 180.000,B 0.000,C 180.000} C_DIS
LIN {X 74.998,Y 40.212,Z 70.000,A 180.000,B 0.000,C 180.000} C_DIS
LIN {X 66.460,Y 43.092,Z 70.000,A 180.000,B 0.000,C 180.000} C_DIS
; Link Move Starts
LIN {X 66.162,Y 43.193,Z 70.000,A 180.000,B 0.000,C 180.000} C_DIS
LIN {X 65.863,Y 43.294,Z 69.999,A 180.000,B 0.000,C 180.000} C_DIS
LIN {X 65.565,Y 43.394,Z 69.998,A 180.000,B 0.000,C 180.000} C_DIS
LIN {X 65.267,Y 43.495,Z 69.996,A 180.000,B 0.000,C 180.000} C_DIS
LIN {X 64.968,Y 43.596,Z 69.994,A 180.000,B 0.000,C 180.000} C_DIS
LIN {X 64.670,Y 43.696,Z 69.991,A 180.000,B 0.000,C 180.000} C_DIS
LIN {X 64.371,Y 43.797,Z 69.988,A 180.000,B 0.000,C 180.000} C_DIS
LIN {X 64.073,Y 43.898,Z 69.985,A 180.000,B 0.000,C 180.000} C_DIS
LIN {X 63.774,Y 43.999,Z 69.981,A 180.000,B 0.000,C 180.000} C_DIS
LIN {X 63.476,Y 44.099,Z 69.977,A 180.000,B 0.000,C 180.000} C_DIS
LIN {X 63.177,Y 44.200,Z 69.972,A 180.000,B 0.000,C 180.000} C_DIS
LIN {X 63.028,Y 44.250,Z 69.969,A 180.000,B 0.000,C 180.000} C_DIS
LIN {X 62.879,Y 44.301,Z 69.967,A 180.000,B 0.000,C 180.000} C_DIS
LIN {X 62.729,Y 44.351,Z 69.964,A 180.000,B 0.000,C 180.000} C_DIS
LIN {X 62.580,Y 44.401,Z 69.961,A 180.000,B 0.000,C 180.000} C_DIS
LIN {X 62.431,Y 44.452,Z 69.959,A 180.000,B 0.000,C 180.000} C_DIS
LIN {X 62.282,Y 44.502,Z 69.956,A 180.000,B 0.000,C 180.000} C_DIS
LIN {X 62.133,Y 44.552,Z 69.952,A 180.000,B 0.000,C 180.000} C_DIS
LIN {X 61.983,Y 44.603,Z 69.949,A 180.000,B 0.000,C 180.000} C_DIS
LIN {X 61.834,Y 44.653,Z 69.946,A 180.000,B 0.000,C 180.000} C_DIS
LIN {X 61.685,Y 44.703,Z 69.943,A 180.000,B 0.000,C 180.000} C_DIS
LIN {X 61.536,Y 44.754,Z 69.939,A 180.000,B 0.000,C 180.000} C_DIS
LIN {X 61.386,Y 44.804,Z 69.936,A 180.000,B 0.000,C 180.000} C_DIS
LIN {X 61.237,Y 44.854,Z 69.932,A 180.000,B 0.000,C 180.000} C_DIS
LIN {X 61.088,Y 44.905,Z 69.928,A 180.000,B 0.000,C 180.000} C_DIS
LIN {X 60.939,Y 44.955,Z 69.925,A 180.000,B 0.000,C 180.000} C_DIS
LIN {X 60.789,Y 45.005,Z 69.921,A 180.000,B 0.000,C 180.000} C_DIS
LIN {X 60.640,Y 45.056,Z 69.917,A 180.000,B 0.000,C 180.000} C_DIS
LIN {X 60.491,Y 45.106,Z 69.913,A 180.000,B 0.000,C 180.000} C_DIS
LIN {X 60.342,Y 45.156,Z 69.909,A 180.000,B 0.000,C 180.000} C_DIS
LIN {X 60.192,Y 45.207,Z 69.905,A 180.000,B 0.000,C 180.000} C_DIS
LIN {X 60.043,Y 45.257,Z 69.900,A 180.000,B 0.000,C 180.000} C_DIS
LIN {X 59.894,Y 45.307,Z 69.896,A 180.000,B 0.000,C 180.000} C_DIS
LIN {X 59.745,Y 45.358,Z 69.892,A 180.000,B 0.000,C 180.000} C_DIS
LIN {X 59.596,Y 45.408,Z 69.887,A 180.000,B 0.000,C 180.000} C_DIS
LIN {X 59.446,Y 45.459,Z 69.883,A 180.000,B 0.000,C 180.000} C_DIS
LIN {X 59.297,Y 45.509,Z 69.878,A 180.000,B 0.000,C 180.000} C_DIS
LIN {X 59.148,Y 45.559,Z 69.873,A 180.000,B 0.000,C 180.000} C_DIS
LIN {X 58.999,Y 45.610,Z 69.869,A 180.000,B 0.000,C 180.000} C_DIS
LIN {X 58.849,Y 45.660,Z 69.864,A 180.000,B 0.000,C 180.000} C_DIS
LIN {X 58.700,Y 45.710,Z 69.859,A 180.000,B 0.000,C 180.000} C_DIS
LIN {X 58.551,Y 45.761,Z 69.854,A 180.000,B 0.000,C 180.000} C_DIS
LIN {X 58.476,Y 45.786,Z 69.851,A 180.000,B 0.000,C 180.000} C_DIS
LIN {X 58.402,Y 45.811,Z 69.849,A 180.000,B 0.000,C 180.000} C_DIS
LIN {X 58.327,Y 45.836,Z 69.846,A 180.000,B 0.000,C 180.000} C_DIS
LIN {X 58.252,Y 45.861,Z 69.844,A 180.000,B 0.000,C 180.000} C_DIS
LIN {X 58.178,Y 45.886,Z 69.841,A 180.000,B 0.000,C 180.000} C_DIS
LIN {X 58.103,Y 45.912,Z 69.839,A 180.000,B 0.000,C 180.000} C_DIS
LIN {X 58.029,Y 45.937,Z 69.836,A 180.000,B 0.000,C 180.000} C_DIS
LIN {X 57.879,Y 45.987,Z 69.831,A 180.000,B 0.000,C 180.000} C_DIS
LIN {X 57.730,Y 46.037,Z 69.825,A 180.000,B 0.000,C 180.000} C_DIS
LIN {X 57.581,Y 46.088,Z 69.820,A 180.000,B 0.000,C 180.000} C_DIS
LIN {X 57.432,Y 46.138,Z 69.815,A 180.000,B 0.000,C 180.000} C_DIS
LIN {X 57.282,Y 46.189,Z 69.809,A 180.000,B 0.000,C 180.000} C_DIS
LIN {X 57.208,Y 46.214,Z 69.807,A 180.000,B 0.000,C 180.000} C_DIS
LIN {X 57.059,Y 46.264,Z 69.801,A 180.000,B 0.000,C 180.000} C_DIS
LIN {X 56.835,Y 46.340,Z 69.793,A 180.000,B 0.000,C 180.000} C_DIS
LIN {X 56.685,Y 46.390,Z 69.787,A 180.000,B 0.000,C 180.000} C_DIS
LIN {X 56.611,Y 46.415,Z 69.785,A 180.000,B 0.000,C 180.000} C_DIS
LIN {X 56.462,Y 46.465,Z 69.779,A 180.000,B 0.000,C 180.000} C_DIS
LIN {X 56.238,Y 46.541,Z 69.771,A 180.000,B 0.000,C 180.000} C_DIS
LIN {X 56.088,Y 46.591,Z 69.765,A 180.000,B 0.000,C 180.000} C_DIS
LIN {X 56.014,Y 46.616,Z 69.763,A 180.000,B 0.000,C 180.000} C_DIS
LIN {X 55.865,Y 46.667,Z 69.757,A 180.000,B 0.000,C 180.000} C_DIS
LIN {X 55.641,Y 46.742,Z 69.749,A 180.000,B 0.000,C 180.000} C_DIS
LIN {X 55.492,Y 46.793,Z 69.743,A 180.000,B 0.000,C 180.000} C_DIS
LIN {X 55.417,Y 46.818,Z 69.741,A 180.000,B 0.000,C 180.000} C_DIS
LIN {X 55.268,Y 46.868,Z 69.735,A 180.000,B 0.000,C 180.000} C_DIS
LIN {X 55.044,Y 46.944,Z 69.727,A 180.000,B 0.000,C 180.000} C_DIS
LIN {X 54.895,Y 46.994,Z 69.721,A 180.000,B 0.000,C 180.000} C_DIS
LIN {X 54.820,Y 47.019,Z 69.719,A 180.000,B 0.000,C 180.000} C_DIS
LIN {X 54.671,Y 47.070,Z 69.713,A 180.000,B 0.000,C 180.000} C_DIS
LIN {X 54.223,Y 47.221,Z 69.697,A 180.000,B 0.000,C 180.000} C_DIS
LIN {X 54.074,Y 47.271,Z 69.691,A 180.000,B 0.000,C 180.000} C_DIS
LIN {X 53.626,Y 47.422,Z 69.675,A 180.000,B 0.000,C 180.000} C_DIS
LIN {X 53.477,Y 47.472,Z 69.669,A 180.000,B 0.000,C 180.000} C_DIS
LIN {X 52.955,Y 47.649,Z 69.650,A 180.000,B 0.000,C 180.000} C_DIS
LIN {X 52.507,Y 47.800,Z 69.633,A 180.000,B 0.000,C 180.000} C_DIS
LIN {X 52.358,Y 47.850,Z 69.628,A 180.000,B 0.000,C 180.000} C_DIS
LIN {X 51.910,Y 48.001,Z 69.611,A 180.000,B 0.000,C 180.000} C_DIS
LIN {X 51.761,Y 48.051,Z 69.606,A 180.000,B 0.000,C 180.000} C_DIS
LIN {X 51.014,Y 48.303,Z 69.578,A 180.000,B 0.000,C 180.000} C_DIS
LIN {X 50.641,Y 48.429,Z 69.565,A 180.000,B 0.000,C 180.000} C_DIS
LIN {X 50.194,Y 48.580,Z 69.548,A 180.000,B 0.000,C 180.000} C_DIS
LIN {X 48.477,Y 49.159,Z 69.485,A 180.000,B 0.000,C 180.000} C_DIS
LIN {X 45.642,Y 50.115,Z 69.380,A 180.000,B 0.000,C 180.000} C_DIS
LIN {X 45.493,Y 50.166,Z 69.375,A 180.000,B 0.000,C 180.000} C_DIS
LIN {X 45.418,Y 50.191,Z 69.372,A 180.000,B 0.000,C 180.000} C_DIS
LIN {X 45.344,Y 50.218,Z 69.369,A 180.000,B 0.000,C 180.000} C_DIS
LIN {X 45.271,Y 50.248,Z 69.367,A 180.000,B 0.000,C 180.000} C_DIS
LIN {X 45.199,Y 50.280,Z 69.364,A 180.000,B 0.000,C 180.000} C_DIS
LIN {X 45.128,Y 50.314,Z 69.361,A 180.000,B 0.000,C 180.000} C_DIS
LIN {X 45.058,Y 50.351,Z 69.358,A 180.000,B 0.000,C 180.000} C_DIS
LIN {X 44.990,Y 50.389,Z 69.356,A 180.000,B 0.000,C 180.000} C_DIS
LIN {X 44.922,Y 50.430,Z 69.353,A 180.000,B 0.000,C 180.000} C_DIS
LIN {X 44.856,Y 50.473,Z 69.350,A 180.000,B 0.000,C 180.000} C_DIS
LIN {X 44.792,Y 50.518,Z 69.347,A 180.000,B 0.000,C 180.000} C_DIS
LIN {X 44.728,Y 50.564,Z 69.345,A 180.000,B 0.000,C 180.000} C_DIS
LIN {X 44.667,Y 50.613,Z 69.342,A 180.000,B 0.000,C 180.000} C_DIS
LIN {X 44.606,Y 50.664,Z 69.339,A 180.000,B 0.000,C 180.000} C_DIS
LIN {X 44.548,Y 50.717,Z 69.336,A 180.000,B 0.000,C 180.000} C_DIS
LIN {X 44.491,Y 50.771,Z 69.334,A 180.000,B 0.000,C 180.000} C_DIS
LIN {X 44.436,Y 50.827,Z 69.331,A 180.000,B 0.000,C 180.000} C_DIS
LIN {X 44.382,Y 50.885,Z 69.328,A 180.000,B 0.000,C 180.000} C_DIS
LIN {X 44.331,Y 50.945,Z 69.325,A 180.000,B 0.000,C 180.000} C_DIS
LIN {X 44.281,Y 51.006,Z 69.323,A 180.000,B 0.000,C 180.000} C_DIS
LIN {X 44.234,Y 51.069,Z 69.320,A 180.000,B 0.000,C 180.000} C_DIS
LIN {X 44.188,Y 51.133,Z 69.317,A 180.000,B 0.000,C 180.000} C_DIS
LIN {X 44.145,Y 51.199,Z 69.314,A 180.000,B 0.000,C 180.000} C_DIS
LIN {X 44.103,Y 51.266,Z 69.312,A 180.000,B 0.000,C 180.000} C_DIS
LIN {X 44.064,Y 51.334,Z 69.309,A 180.000,B 0.000,C 180.000} C_DIS
LIN {X 44.026,Y 51.403,Z 69.306,A 180.000,B 0.000,C 180.000} C_DIS
LIN {X 43.991,Y 51.474,Z 69.303,A 180.000,B 0.000,C 180.000} C_DIS
LIN {X 43.959,Y 51.545,Z 69.301,A 180.000,B 0.000,C 180.000} C_DIS
LIN {X 43.928,Y 51.618,Z 69.298,A 180.000,B 0.000,C 180.000} C_DIS
LIN {X 43.900,Y 51.692,Z 69.295,A 180.000,B 0.000,C 180.000} C_DIS
LIN {X 43.874,Y 51.766,Z 69.292,A 180.000,B 0.000,C 180.000} C_DIS
LIN {X 43.851,Y 51.841,Z 69.290,A 180.000,B 0.000,C 180.000} C_DIS
LIN {X 43.830,Y 51.917,Z 69.287,A 180.000,B 0.000,C 180.000} C_DIS
LIN {X 43.811,Y 51.994,Z 69.284,A 180.000,B 0.000,C 180.000} C_DIS
LIN {X 43.795,Y 52.071,Z 69.281,A 180.000,B 0.000,C 180.000} C_DIS
LIN {X 43.781,Y 52.148,Z 69.279,A 180.000,B 0.000,C 180.000} C_DIS
LIN {X 43.769,Y 52.226,Z 69.276,A 180.000,B 0.000,C 180.000} C_DIS
LIN {X 43.760,Y 52.304,Z 69.273,A 180.000,B 0.000,C 180.000} C_DIS
LIN {X 43.754,Y 52.383,Z 69.270,A 180.000,B 0.000,C 180.000} C_DIS
LIN {X 43.750,Y 52.461,Z 69.268,A 180.000,B 0.000,C 180.000} C_DIS
LIN {X 43.748,Y 52.540,Z 69.265,A 180.000,B 0.000,C 180.000} C_DIS
LIN {X 43.749,Y 52.619,Z 69.262,A 180.000,B 0.000,C 180.000} C_DIS
LIN {X 43.753,Y 52.698,Z 69.259,A 180.000,B 0.000,C 180.000} C_DIS
LIN {X 43.759,Y 52.776,Z 69.257,A 180.000,B 0.000,C 180.000} C_DIS
LIN {X 43.767,Y 52.855,Z 69.254,A 180.000,B 0.000,C 180.000} C_DIS
LIN {X 43.778,Y 52.933,Z 69.251,A 180.000,B 0.000,C 180.000} C_DIS
LIN {X 43.791,Y 53.010,Z 69.248,A 180.000,B 0.000,C 180.000} C_DIS
LIN {X 43.807,Y 53.087,Z 69.246,A 180.000,B 0.000,C 180.000} C_DIS
LIN {X 43.825,Y 53.164,Z 69.243,A 180.000,B 0.000,C 180.000} C_DIS
LIN {X 43.846,Y 53.240,Z 69.240,A 180.000,B 0.000,C 180.000} C_DIS
LIN {X 43.869,Y 53.315,Z 69.237,A 180.000,B 0.000,C 180.000} C_DIS
LIN {X 43.894,Y 53.390,Z 69.235,A 180.000,B 0.000,C 180.000} C_DIS
LIN {X 43.944,Y 53.539,Z 69.229,A 180.000,B 0.000,C 180.000} C_DIS
LIN {X 44.019,Y 53.763,Z 69.221,A 180.000,B 0.000,C 180.000} C_DIS
LIN {X 44.070,Y 53.912,Z 69.215,A 180.000,B 0.000,C 180.000} C_DIS
LIN {X 44.095,Y 53.987,Z 69.213,A 180.000,B 0.000,C 180.000} C_DIS
LIN {X 44.145,Y 54.136,Z 69.207,A 180.000,B 0.000,C 180.000} C_DIS
LIN {X 44.221,Y 54.360,Z 69.199,A 180.000,B 0.000,C 180.000} C_DIS
LIN {X 44.271,Y 54.509,Z 69.193,A 180.000,B 0.000,C 180.000} C_DIS
LIN {X 44.372,Y 54.808,Z 69.182,A 180.000,B 0.000,C 180.000} C_DIS
LIN {X 44.422,Y 54.957,Z 69.177,A 180.000,B 0.000,C 180.000} C_DIS
LIN {X 44.472,Y 55.106,Z 69.172,A 180.000,B 0.000,C 180.000} C_DIS
LIN {X 44.523,Y 55.256,Z 69.166,A 180.000,B 0.000,C 180.000} C_DIS
LIN {X 44.548,Y 55.330,Z 69.164,A 180.000,B 0.000,C 180.000} C_DIS
LIN {X 44.573,Y 55.405,Z 69.161,A 180.000,B 0.000,C 180.000} C_DIS
LIN {X 44.598,Y 55.479,Z 69.159,A 180.000,B 0.000,C 180.000} C_DIS
LIN {X 44.624,Y 55.554,Z 69.156,A 180.000,B 0.000,C 180.000} C_DIS
LIN {X 44.649,Y 55.629,Z 69.154,A 180.000,B 0.000,C 180.000} C_DIS
LIN {X 44.674,Y 55.703,Z 69.151,A 180.000,B 0.000,C 180.000} C_DIS
LIN {X 44.699,Y 55.778,Z 69.149,A 180.000,B 0.000,C 180.000} C_DIS
LIN {X 44.749,Y 55.927,Z 69.144,A 180.000,B 0.000,C 180.000} C_DIS
LIN {X 44.800,Y 56.076,Z 69.139,A 180.000,B 0.000,C 180.000} C_DIS
LIN {X 44.850,Y 56.226,Z 69.134,A 180.000,B 0.000,C 180.000} C_DIS
LIN {X 44.900,Y 56.375,Z 69.129,A 180.000,B 0.000,C 180.000} C_DIS
LIN {X 44.951,Y 56.524,Z 69.124,A 180.000,B 0.000,C 180.000} C_DIS
LIN {X 45.001,Y 56.673,Z 69.120,A 180.000,B 0.000,C 180.000} C_DIS
LIN {X 45.051,Y 56.822,Z 69.115,A 180.000,B 0.000,C 180.000} C_DIS
LIN {X 45.102,Y 56.972,Z 69.111,A 180.000,B 0.000,C 180.000} C_DIS
LIN {X 45.152,Y 57.121,Z 69.106,A 180.000,B 0.000,C 180.000} C_DIS
LIN {X 45.202,Y 57.270,Z 69.102,A 180.000,B 0.000,C 180.000} C_DIS
LIN {X 45.253,Y 57.419,Z 69.097,A 180.000,B 0.000,C 180.000} C_DIS
LIN {X 45.303,Y 57.569,Z 69.093,A 180.000,B 0.000,C 180.000} C_DIS
LIN {X 45.354,Y 57.718,Z 69.089,A 180.000,B 0.000,C 180.000} C_DIS
LIN {X 45.404,Y 57.867,Z 69.085,A 180.000,B 0.000,C 180.000} C_DIS
LIN {X 45.454,Y 58.016,Z 69.081,A 180.000,B 0.000,C 180.000} C_DIS
LIN {X 45.505,Y 58.166,Z 69.077,A 180.000,B 0.000,C 180.000} C_DIS
LIN {X 45.555,Y 58.315,Z 69.073,A 180.000,B 0.000,C 180.000} C_DIS
LIN {X 45.605,Y 58.464,Z 69.070,A 180.000,B 0.000,C 180.000} C_DIS
LIN {X 45.656,Y 58.613,Z 69.066,A 180.000,B 0.000,C 180.000} C_DIS
LIN {X 45.706,Y 58.763,Z 69.062,A 180.000,B 0.000,C 180.000} C_DIS
LIN {X 45.756,Y 58.912,Z 69.059,A 180.000,B 0.000,C 180.000} C_DIS
LIN {X 45.807,Y 59.061,Z 69.056,A 180.000,B 0.000,C 180.000} C_DIS
LIN {X 45.857,Y 59.210,Z 69.052,A 180.000,B 0.000,C 180.000} C_DIS
LIN {X 45.907,Y 59.360,Z 69.049,A 180.000,B 0.000,C 180.000} C_DIS
LIN {X 45.958,Y 59.509,Z 69.046,A 180.000,B 0.000,C 180.000} C_DIS
LIN {X 46.008,Y 59.658,Z 69.043,A 180.000,B 0.000,C 180.000} C_DIS
LIN {X 46.058,Y 59.807,Z 69.040,A 180.000,B 0.000,C 180.000} C_DIS
LIN {X 46.109,Y 59.956,Z 69.037,A 180.000,B 0.000,C 180.000} C_DIS
LIN {X 46.159,Y 60.106,Z 69.034,A 180.000,B 0.000,C 180.000} C_DIS
LIN {X 46.209,Y 60.255,Z 69.032,A 180.000,B 0.000,C 180.000} C_DIS
LIN {X 46.260,Y 60.404,Z 69.029,A 180.000,B 0.000,C 180.000} C_DIS
LIN {X 46.310,Y 60.553,Z 69.027,A 180.000,B 0.000,C 180.000} C_DIS
LIN {X 46.411,Y 60.852,Z 69.022,A 180.000,B 0.000,C 180.000} C_DIS
